// POUs/System/SystemInfo
{attribute 'no_check'}
//Provides all information of PlcAppSystemInfo plus addtional infos like time stamps from various source and in different formats
//
//PlcAppSystemInfo -> https://infosys.beckhoff.com/english.php?content=../content/1033/globaldatatypes/9007199969559691.html&id=7934476013631172214
//TwimCAT time sources -> https://infosys.beckhoff.com/english.php?content=../content/1033/ethercatsystem/2469114379.html&id=
//
FUNCTION_BLOCK SystemInfo
VAR_OUTPUT CONSTANT
{attribute 'displaymode':='binary'}
	OPTION_US_DATE_FORMAT									:	BYTE := 2#0000_0001; //Enable US date format in time stamp - mm/dd/yy
{attribute 'displaymode':='binary'}
	OPTION_US_TIME_FORMAT									:	BYTE := 2#0000_0010; //Enable time in US format - AM/PM vs 24h
{attribute 'displaymode':='binary'} 
	OPTION_TIME_STR_ADD_MS									:	BYTE := 2#0000_0100; //Add ms to time string 
{attribute 'displaymode':='binary'} 
	OPTION_DISABLE_DEV_IDENT								:	BYTE := 2#0000_1000; //Disable to read device identification during boot up (Call FB_GetDeviceIdentificationEx)
END_VAR                     								
VAR_INPUT                   						
	Enable													:	BOOL := TRUE; //Enable function block
	ResetTrig												:	BOOL := FALSE; //Reset Old boot data fault signal
	RtcSyncCylce											:	DWORD := 60; //in seconds - see documentation for "FB_LocalSystemTime"
	KeepOutputsOnBP 										: 	BOOL := FALSE; //The flag can be set to avoid that the outputs are zero-filled if a breakpoint is reached. The task keeps running. Only the execution of PLC code is interrupted.
{attribute 'displaymode':='binary'}
	Options													:	BYTE := 2#0000_0000; //option constants are alreay predefined, so they can accordingly be passed symbolically to the block 
	DateStrSeperator										:	STRING(1) := '/';
END_VAR
VAR_OUTPUT
//PlcAppSystemInfo and cycle time inforamtion from caller task 
	ObjId													: 	OTCID; //Object ID of the PLC project instance
	AdsPort 												: 	UINT; //ADS port of PLC application 
	TComSrvPtr 												: 	ITComObjectServer; // Pointer to TcCOM Object Server 
	AppName													: 	STRING(63); //TwinCAT generated name containing the port number. 
	ProjectName 											: 	STRING(63); //The name of the PLC project. 
	AppTimestampDT											:	DT; //Date and time of application start 
	AppTimestamp											:	STRING(25);	//Date and time of application start in string format
	TaskIndex												:	INT ; //Task index of SysInfo caller
	TaskCnt													: 	UDINT; //The number of tasks in the actual runtime system
	
	Flags 													: 	DWORD; //Boot flags
	LicensesPending 										: 	BOOL;
	BSODOccured 											: 	BOOL;										
	BootDataLoaded											: 	BOOL;//PERSISTENT variables: LOADED (without error)
	OldBootData												: 	BOOL; //PERSISTENT variables: INVALID (the back-up copy was loaded, since no valid data was present)
	NoBootDataLoaded										:	BOOL; //Error no boot data loaded
//	PersistentStatus 										: 	EPlcPersistentStatus;

	LoggedIn												:	BOOL;
	ShutdownInProgress 										: 	BOOL;	
	OnlineChangeCount										: 	UDINT; //The number of online changes made since the last complete download.
	OnlineChange											:	BOOL; //Online change count changed since last plc cycle

{attribute 'displaymode':='hex'}
	CpuCounter												:	ULINT;
	CycleTime         										: 	UDINT;//Cylce time read from PlcAppSystemInfo in multiples of 100 ns.
	CycleTimeNS         									: 	UDINT;//Cylce time in nanoseconds
	CycleTimeT       										: 	TIME; //Cycle time in time format
	CycleTimeLT       										: 	LTIME; //Cycle time in ltime format
	CycleTimeFloat											:	LREAL;//Cycle time in float format <s.ms>

	DevIdentValid											:	BOOL;
	pDevIdent												:	POINTER TO ST_DeviceIdentificationEx := ADR(InstGetDevIdent.stDevIdent);
	
//General	
	TimezoneId												: 	E_TimeZoneID;
	TimeZoneInfo											:	ST_TimeZoneInformation; //Provides actual time zone and bias from local time to UTC e.g. UTC=MEC-01:00 (-60min from lcoal MEZ in Standard time to UTC)
	MonthDays												:	WORD;
	LeapYear												:	BOOL;
	DayOfYear												:	WORD;
	WeekOfYear												:	WORD;
	UtcTimeFT												:	Tc2_Utilities.T_FILETIME; //Current UTC System/TwinCAT time T_FILETIME format, structure representing a 64-bit value with the a number of 100-nanosecond intervals since January 1, 1601 (UTC) (dwLowDateTime : DWORD / dwHighDateTime : DWORD)
//	UtcTimeFT												:	Tc2_Utilities.T_FILETIME64; //Current UTC System/TwinCAT time T_FILETIME format, structure representing a 64-bit value with the a number of 100-nanosecond intervals since January 1, 1601 (UTC) (dwLowDateTime : DWORD / dwHighDateTime : DWORD)
	UtcTimeSTRUCT											:	Tc2_Utilities.TIMESTRUCT; //Current UTC System/TwinCAT time in TIMESTRUCT format
	UtcTimezoneBias											:	DINT;   //Bias from UTC to local time in minutes e.g. MEZ=UTC+01:00 (60min)  
	TimeDT													:	DATE_AND_TIME;	//Current time in DATE_AND_TIME format: DT#1970-01-01-00:00 -> DT#2106-02-06-06:28:15
//	TimeLDT													:	LDATE_AND_TIME;	//Current time in 64bit LDATE_AND_TIME format: DT#1970-01-01-00:00 -> DT#2262-4-10-23:59:59.99999999
	TimeTOD													:	TOD; //Current time in TOD format, range from TOD#00:00 -> TOD#1193:02:47.295
	TimeFT													:	Tc2_Utilities.T_FILETIME; //Current time in T_FILETIME format, structur representing a 64-bit value with the a number of 100-nanosecond intervals since January 1, 1601 (UTC) (dwLowDateTime : DWORD / dwHighDateTime : DWORD)
//	TimeFT													:	Tc2_Utilities.T_FILETIME64; //Current time in T_FILETIME format, structur representing a 64-bit value with the a number of 100-nanosecond intervals since January 1, 1601 (UTC) (dwLowDateTime : DWORD / dwHighDateTime : DWORD)
	TimeSTRUCT												:	Tc2_Utilities.TIMESTRUCT; //Current time in TIMESTRUCT format
	Datestamp												:	DATE; //D#1970-01-01 -> D#2106-02-06
	DateStr													:	STRING(15);	(* dd.mm.jj or mm.dd.jj *)	
	TimeStr													:	STRING(15);	(* hh:mm:ss.xxx or hh:mm:ss.xxxPM/AM *)
	TimeStamp												:	STRING(25); (* DateStr + TimeStr *)	
	TimeStamp2												:	STRING(25); (* YYYY-MM-DDTHHMMSS for example YYYY-MM-DD_HHMMSS_Name.txt *)
	TimeStamp3												:	STRING(25); (* YYYY-MM-DD-hh:mm:ss.xxx *)
	DateStrISO												:	STRING(15);	(* jjjj-mm-dd *)
	TimeStrISO												:	STRING(15);	(* hh:mm:ss *)
	TimeStrISO2												:	STRING(15);	(* hh:mm:ss.xxx *)	
	TimeStampIso											:	STRING(30);	(* jjjj-mm-dd'T'hh:mm:ss.xxx local time*)	
//	TimeStampIsoZulu										:	STRING(30);	(* jjjj-mm-dd'T'hh:mm:ss.xmsZ - Iso timestamp in UTC (ZULU)*)	
//	TimeStampIsoUtc											:	STRING(30);	(* jjjj-mm-dd'T'hh:mm:ss.xms+mm:ss - Iso timestamp with UTC offset *)	

	TimeStampStartup										:	DATE_AND_TIME; //Timestamp of startup
	DCTime													:	Tc2_EtherCAT.T_DCTIME64; //Current TwinCAT distributed clock time in 64-bit T_DCTIME64 format. The smallest unit is a nanosecond.
	DCTimeSTRUCT											:	Tc2_Utilities.TIMESTRUCT;//Current TwinCAT distributed clock time in TIMESTRUCT format
//	SysTimeFT												:	Tc2_Utilities.T_FILETIME64; //Current UTC System/TwinCAT time T_FILETIME format, structure representing a 64-bit value with the a number of 100-nanosecond intervals since January 1, 1601 (UTC) (dwLowDateTime : DWORD / dwHighDateTime : DWORD)
	SysTimeFT												:	Tc2_Utilities.T_FILETIME; //Current UTC System/TwinCAT time T_FILETIME format, structure representing a 32-bit value since January 1, 1601 (UTC) (dwLowDateTime : DWORD / dwHighDateTime : DWORD)
	SysTimeSTRUCT											:	Tc2_Utilities.TIMESTRUCT; //Current UTC System/TwinCAT time in TIMESTRUCT format
	
END_VAR
VAR
	(* Inst. Get Taskindex *)
	InstGETCURTASKINDEX										: 	GETCURTASKINDEX;
	InstLocalSystemTime										:	FB_LocalSystemTime;
	InstNtSetLocalTime										:	NT_SetLocalTime := (NETID := '', TMOUT := DEFAULT_ADS_TIMEOUT);
	InstTimeZoneInfo										:	FB_GetTimeZoneInformation;
	InstCpuCouter											:	GETCPUCOUNTER;
	InstSystemTime											:	GetSystemTime;
	
	
	InstGetDevIdent											:	FB_GetDeviceIdentificationEx;
	_OnlineChangeCount										: 	UDINT; 
	_sec													:	WORD;
	_hour													:	WORD;
	_day													:	WORD;
	_Init													:	BOOL;
END_VAR

	(* Evaluate the PlcAppSystemInfo and and get sytstem timestamp					*)
	(********************************************************************************)
	
(* Get Current Task Index ************************************************************************)
	IF InstGETCURTASKINDEX.index = 0 then InstGETCURTASKINDEX(index => TaskIndex); END_IF

(* Read System Info Current Task *****************************************************************)	
	(* Get static information and boot error messages *)
	IF TwinCAT_SystemInfoVarList._TaskInfo[InstGETCURTASKINDEX.Index].FirstCycle 
	THEN
		AppTimestampDT										:= TwinCAT_SystemInfoVarList._AppInfo.AppTimestamp;
		AppTimestamp										:= DT_TO_STRING(AppTimestampDT);
		AppTimestamp										:= DELETE(AppTimestamp,3,1);
			
		TaskIndex											:= InstGETCURTASKINDEX.Index;
		TaskCnt 											:= TwinCAT_SystemInfoVarList._AppInfo.TaskCnt;
		
		ObjId												:= TwinCAT_SystemInfoVarList._AppInfo.ObjId;
		AppName												:= TwinCAT_SystemInfoVarList._AppInfo.AppName;	
		ProjectName											:= TwinCAT_SystemInfoVarList._AppInfo.ProjectName;	
		AdsPort												:= TwinCAT_SystemInfoVarList._AppInfo.AdsPort;	
			
		Flags												:= TwinCAT_SystemInfoVarList._AppInfo.Flags;
//		PersistentStatus									:= TwinCAT_SystemInfoVarList._AppInfo.PersistentStatus;
		
		BootDataLoaded										:= TwinCAT_SystemInfoVarList._AppInfo.BootDataLoaded;
		OldBootData											:= TwinCAT_SystemInfoVarList._AppInfo.OldBootData;
		NoBootDataLoaded									:= NOT BootDataLoaded AND NOT OldBootData;
		BSODOccured 										:= TwinCAT_SystemInfoVarList._AppInfo.BSODOccured;
		
		CycleTime         									:= TwinCAT_SystemInfoVarList._TaskInfo[TaskIndex].CycleTime;
		CycleTimeNS         								:= TwinCAT_SystemInfoVarList._TaskInfo[TaskIndex].CycleTime * 100;
		CycleTimeT											:= LREAL_TO_TIME(UDINT_TO_LREAL(CycleTime) * 0.0001 );
		CycleTimeLT											:= TO_LTIME(CycleTimeNS);	
		CycleTimeFloat										:= (UDINT_TO_LREAL(CycleTime) * 0.0001 / 1000.0);	
		
	ELSIF ResetTrig
	THEN
		resetBootInfo();
	ELSIF NOT Enable
	THEN
		RETURN;
	END_IF
	
	OnlineChangeCount										:= TwinCAT_SystemInfoVarList._AppInfo.OnlineChangeCnt;
	OnlineChange											:= _OnlineChangeCount <> OnlineChangeCount;
	_OnlineChangeCount										:= OnlineChangeCount;
	LoggedIn 												:= TwinCAT_SystemInfoVarList._AppInfo.LoggedIn;
	ShutdownInProgress 										:= TwinCAT_SystemInfoVarList._AppInfo.ShutdownInProgress;
	LicensesPending 										:= TwinCAT_SystemInfoVarList._AppInfo.LicensesPending;
	TComSrvPtr												:= TwinCAT_SystemInfoVarList._AppInfo.TComSrvPtr;
	TwinCAT_SystemInfoVarList._AppInfo.KeepOutputsOnBP		:= KeepOutputsOnBP;		

(* CPU System counter ****************************************************************************)
	InstCpuCouter(cpuCntLoDW => CpuCounter);	
	MEMCPY(ADR(CpuCounter) + SIZEOF(InstCpuCouter.cpuCntHiDW),ADR(InstCpuCouter.cpuCntHiDW),SIZEOF(InstCpuCouter.cpuCntHiDW));
	
(* Get device identification structure ***********************************************************)
	InstGetDevIdent(
		bExecute	:= NOT Options.3, 
		tTimeout	:= , 
		sNetId		:= , 
		bBusy		=> , 
		bError		=> , 
		nErrorID	=> , 
		stDevIdent	=> );	
	pDevIdent												:= ADR(InstGetDevIdent.stDevIdent);
	IF NOT InstGetDevIdent.bBusy
	THEN
		DevIdentValid										:= NOT InstGetDevIdent.bError;
		
		IF InstGetDevIdent.bError AND ResetTrig
		THEN
			InstGetDevIdent(bExecute := FALSE);			
		END_IF
	ELSE	
		DevIdentValid										:= FALSE;
	END_IF
	
(* Read timezone information every day time ******************************************************)
	IF Enable AND NOT InstTimeZoneInfo.bExecute
		OR InstTimeZoneInfo.bBusy
	THEN
		InstTimeZoneInfo(
			sNetID	:= , 
			bExecute:= TRUE, 
			tTimeout:= , 
			bBusy	=> , 
			bError	=> , 
			nErrID	=> , 
			tzID	=> TimeZoneId, 
			tzInfo	=> TimeZoneInfo);
		IF NOT InstTimeZoneInfo.bBusy 
		THEN
			CASE TimeZoneId OF 
			eTimeZoneID_Invalid:	UtcTimezoneBias			:= 0;				
			eTimeZoneID_Standard:	UtcTimezoneBias			:= -1 * (TimeZoneInfo.bias + TimeZoneInfo.standardBias);
			eTimeZoneID_Daylight:	UtcTimezoneBias			:= -1 * (TimeZoneInfo.bias + TimeZoneInfo.daylightBias);
			ELSE //eTimeZoneID_Unknown:		
				UtcTimezoneBias								:= 0;	
			END_CASE
		END_IF
	ELSIF NOT Enable AND InstTimeZoneInfo.bExecute 
		OR InstTimeZoneInfo.bError AND ResetTrig
	THEN
		InstTimeZoneInfo(bExecute:= FALSE);
	END_IF
		
(* Actual EtherCAT DC time in DCTIME64 format ****************************************************************)
	DCTime													:= F_GetActualDcTime64();
	DCTimeSTRUCT											:= DCTIME64_TO_SYSTEMTIME(DCTime);

(* Get TwinCAT/system time according to system time zone initialized during TC start ******************************************************)
	InstSystemTime(timeHiDW => UtcTimeFT.dwHighDateTime,timeLoDW => UtcTimeFT.dwLowDateTime );
	SysTimeSTRUCT											:= FILETIME_TO_SYSTEMTIME(UTCTimeFT);	
	
//	SysTimeFT												:= F_GetSystemTime();	 
//	SysTimeSTRUCT											:= FILETIME64_TO_SYSTEMTIME(UTCTimeFT);	 
	
(* evalutate systemtime ************************************************************************)
	InstLocalSystemTime(
		sNetID		:= '',
		bEnable		:= Enable,
		dwCycle		:= SEL(InstNtSetLocalTime.START, RtcSyncCylce, 1), //Short update cylce to read windows time after it was set
		dwopt		:= (* Default *),
		tTimeout	:= (* Default *),
		bValid		=> ,
		systemTime	=> TimeSTRUCT,
		tzID		=> );

(* Get TwinCAT/system time in UTC Filetime format ******************************************************)
	IF InstLocalSystemTime.bValid 
	THEN				
		//Update cyclic
//		TimeFT												:= SYSTEMTIME_TO_FILETIME64(TimeSTRUCT);
		TimeFT												:= SYSTEMTIME_TO_FILETIME(TimeSTRUCT);
		TimeDT 												:= SYSTEMTIME_TO_DT(TimeSTRUCT);
//		TimeLDT												:= SYSTEMTIME_TO_LDT(TimeSTRUCT);	
		TimeStamp3											:= SYSTEMTIME_TO_STRING(TimeSTRUCT);
		TimeTOD												:= SEL(Options.2 ,TO_TOD(TimeDT)  , DWORD_TO_TOD(TO_DWORD(TO_TOD(TimeDT)) + TimeSTRUCT.wMilliseconds));  
		TimeStrISO											:= DELETE(TO_STRING(TimeTOD),4,1);

		IF TimeSTRUCT.wMilliseconds < 10 
		THEN
			TimeStrISO2 									:= CONCAT(TimeStrISO,CONCAT('.00',WORD_TO_STRING(TimeSTRUCT.wMilliseconds)));
		ELSIF TimeSTRUCT.wMilliseconds < 100
		THEN
			TimeStrISO2 									:= CONCAT(TimeStrISO,CONCAT('.0',WORD_TO_STRING(TimeSTRUCT.wMilliseconds)));			
		ELSE        										
			TimeStrISO2 									:= CONCAT(TimeStrISO,CONCAT('.',WORD_TO_STRING(TimeSTRUCT.wMilliseconds)));	
		END_IF 	
		
		TimeStampISO										:= CONCAT(DateStrISO , CONCAT('T',TimeStrISO2));
				
		UtcTimeFT											:= F_TranslateFileTimeBias(TimeFT,UtcTimezoneBias,TRUE);
		UtcTimeSTRUCT										:= FILETIME_TO_SYSTEMTIME(UTCTimeFT);	
//		UtcTimeFT											:= F_TranslateFileTime64Bias(TimeFT,UtcTimezoneBias,TRUE);
//		UtcTimeSTRUCT										:= FILETIME64_TO_SYSTEMTIME(UTCTimeFT);	

//		TimeStampIsoZulu									:= SYSTEMTIME_TO_ISO8601(UtcTimeSTRUCT,0,FALSE,3);
//		TimeStampIsoZulu									:= CONCAT(DELETE(TimeStampIsoZulu,6,24),'Z');
//		TimeStampIsoUtc										:= SYSTEMTIME_TO_ISO8601(UtcTimeSTRUCT,TO_INT(UtcTimezoneBias),TRUE,3);
	
		//Create time format
		IF Options.1
		THEN (* US time format hh.mm.ss AM/PM ***************)
			IF TimeSTRUCT.wHour < 10 
			THEN
				TimeStr 									:= CONCAT('0',WORD_TO_STRING(TimeSTRUCT.wHour));
			ELSIF TimeSTRUCT.wHour > 12 
			THEN
				TimeStr 									:= WORD_TO_STRING(TimeSTRUCT.wHour - 12);
				IF TimeSTRUCT.wHour - 12 < 10
				THEN
					TimeStr									:= CONCAT('0',TimeStr);
				END_IF
			ELSE         									
				TimeStr 									:= WORD_TO_STRING(TimeSTRUCT.wHour);
			END_IF		                                    
		ELSE  (* Time hh.mm.ss.xxms ***************)          
			IF TimeSTRUCT.wHour < 10                        
			THEN                                            
				TimeStr 									:= CONCAT('0',WORD_TO_STRING(TimeSTRUCT.wHour));
			ELSE        									
				TimeStr 									:= WORD_TO_STRING(TimeSTRUCT.wHour);
			END_IF			
		END_IF
		
		TimeStr 											:= CONCAT(TimeStr,':');
		
		IF TimeSTRUCT.wMinute < 10 
		THEN
			TimeStr 										:= CONCAT(TimeStr,CONCAT('0',WORD_TO_STRING(TimeSTRUCT.wMinute)));
		ELSE
			TimeStr 										:= CONCAT(TimeStr,WORD_TO_STRING(TimeSTRUCT.wMinute));
		END_IF
		
		TimeStr 											:= CONCAT(TimeStr,':');
		
		IF TimeSTRUCT.wSecond < 10 
		THEN
			TimeStr 										:= CONCAT(TimeStr,CONCAT('0',WORD_TO_STRING(TimeSTRUCT.wSecond)));
		ELSE        										
			TimeStr 										:= CONCAT(TimeStr,WORD_TO_STRING(TimeSTRUCT.wSecond));
		END_IF  
												
		IF Options.2
		THEN //add ms to timestamp
			TimeStr 										:= CONCAT(TimeStr,'.');
			TimeStr 										:= CONCAT(TimeStr,WORD_TO_STRING(TimeSTRUCT.wMilliseconds));
		END_IF
		
		IF Options.1
		THEN //US time format
			TimeStr 										:= CONCAT(TimeStr,SEL(TimeSTRUCT.wHour > 12,' AM', ' PM'));
		END_IF
		
		(* TimeStamp Format DE: DD.MM.YY-Stunde:Minute:Sekunde.xxx,*)
		TimeStamp 											:= CONCAT(DateStr,'-');
		TimeStamp 											:= CONCAT(TimeStamp,TimeStr);
		
		IF _hour <> TimeSTRUCT.wHour OR NOT _Init
		THEN
			_Hour											:= TimeSTRUCT.wHour;		
			//Create date in US fromat with seperator / ************************************************
			IF Options.0
			THEN (* Date mm/dd/jj ********************)
				IF TimeSTRUCT.wMonth < 10 
				THEN
					DateStr 								:= CONCAT('0',WORD_TO_STRING(TimeSTRUCT.wMonth));
				ELSE        								
					DateStr 								:= WORD_TO_STRING(TimeSTRUCT.wMonth);
				END_IF		                                
				DateStr 									:= CONCAT(DateStr,DateStrSeperator);
				IF TimeSTRUCT.wDay < 10                     
				THEN                                        
					DateStr 								:= CONCAT(DateStr,CONCAT('0',WORD_TO_STRING(TimeSTRUCT.wDay)));
				ELSE        								
					DateStr 								:= CONCAT(DateStr,WORD_TO_STRING(TimeSTRUCT.wDay));
				END_IF                                      
															
				DateStr 									:= CONCAT(DateStr,DateStrSeperator);
				DateStr 									:= CONCAT(DateStr,RIGHT(WORD_TO_STRING(TimeSTRUCT.wYear),2));		
		                                                    
			ELSE (* Date dd.mm.jj ********************)	    
				IF TimeSTRUCT.wDay < 10                     
				THEN                                        
					DateStr 								:= CONCAT('0',WORD_TO_STRING(TimeSTRUCT.wDay));
				ELSE        								
					DateStr 								:= WORD_TO_STRING(TimeSTRUCT.wDay);
				END_IF                                      
				DateStr 									:= CONCAT(DateStr,DateStrSeperator);
				IF TimeSTRUCT.wMonth < 10                   
				THEN                                        
					DateStr 								:= CONCAT(DateStr,CONCAT('0',WORD_TO_STRING(TimeSTRUCT.wMonth)));
				ELSE        								
					DateStr 								:= CONCAT(DateStr,WORD_TO_STRING(TimeSTRUCT.wMonth));
				END_IF                                      
															
				DateStr 									:= CONCAT(DateStr,DateStrSeperator);
				DateStr 									:= CONCAT(DateStr,RIGHT(WORD_TO_STRING(TimeSTRUCT.wYear),2));	
			END_IF      

			DateStrISO										:= DELETE(TO_STRING(TO_DATE(TimeDT)),2,1);
			
			(* information of year *)                       
			MonthDays										:= F_GetMaxMonthDays(TimeSTRUCT.wYear,TimeSTRUCT.wMonth);
			LeapYear										:= F_YearIsLeapYear(TimeSTRUCT.wYear) ;
			WeekOfYear										:= F_GetWeekOfTheYear(TimeDT);
			DayOfYear										:= F_GetDOYOfYearMonthDay(TimeSTRUCT.wYear,TimeSTRUCT.wMonth,TimeSTRUCT.wDay);
			DateStamp										:= TO_DATE(TimeDT);		
			
			IF NOT _INIT AND_THEN TO_DINT(TimeStampStartup) = 0  
			THEN					
				TimeStampStartup							:= SYSTEMTIME_TO_DT(TimeSTRUCT);
			END_IF
			
			IF NOT InstTimeZoneInfo.bBusy THEN InstTimeZoneInfo(bExecute:= FALSE); END_IF

            _INIT											:= TRUE;            
		END_IF //hour
		
		IF _sec <> TimeSTRUCT.wSecond 
		THEN	
			_sec 											:= TimeSTRUCT.wSecond;
														
			(* TimeStamp2 FileName YYYY-MM-DD_HHMMSS *)
			TimeStamp2										:= CONCAT(DateStrISO , '_');
			IF TimeSTRUCT.wHour < 10                    	
			THEN                                        	
				TimeStamp2 									:= CONCAT(TimeStamp2,CONCAT('0',WORD_TO_STRING(TimeSTRUCT.wHour)));
			ELSE           									
				TimeStamp2 									:= CONCAT(TimeStamp2,WORD_TO_STRING(TimeSTRUCT.wHour));
			END_IF                                      	
			IF TimeSTRUCT.wMinute < 10                  	
			THEN                                        	
				TimeStamp2 									:= CONCAT(TimeStamp2,CONCAT('0',WORD_TO_STRING(TimeSTRUCT.wMinute)));
			ELSE           									
				TimeStamp2 									:= CONCAT(TimeStamp2,WORD_TO_STRING(TimeSTRUCT.wMinute));
			END_IF                                      	
			IF TimeSTRUCT.wSecond < 10                  	
			THEN                                        	
				TimeStamp2 									:= CONCAT(TimeStamp2,CONCAT('0',WORD_TO_STRING(TimeSTRUCT.wSecond)));
			ELSE           									
				TimeStamp2 									:= CONCAT(TimeStamp2,WORD_TO_STRING(TimeSTRUCT.wSecond));
			END_IF
		END_IF //second update
													
	END_IF

(* set system time *****************************************************************************)
	InstNtSetLocalTime(
		NETID		:= , 
		TIMESTR		:= , 
		START		:= , // Start by Methode "SetSysTime" 
		TMOUT		:= , 
		BUSY		=> , 
		ERR			=> ); 
	
	IF InstNtSetLocalTime.START AND NOT InstNtSetLocalTime.BUSY
	THEN //Take care that all timestamp get updated after set a new time
		InstNtSetLocalTime.START							:= FALSE;	
		_Init												:= FALSE;								
	END_IF
	
(**************************************************************************************************)

PROPERTY PUBLIC actDCTimeWithTimezoneBias : T_DCTIME64
GET
actDCTimeWithTimezoneBias							:= F_GetActualDcTime64() + (TO_ULINT(UtcTimezoneBias) * 60 * EC_DCTIME_TICKSPERSEC64);
END_GET
END_PROPERTY

PROPERTY PUBLIC optAddmsToTimeString : BOOL
GET
optAddmsToTimeString := Options.2;
END_GET
SET
Options.2 := optAddmsToTimeString;
END_SET
END_PROPERTY

PROPERTY PUBLIC  optDisableReadDeviceIdentification : BOOL
GET
optDisableReadDeviceIdentification := Options.3;
END_GET
SET
Options.3 := optDisableReadDeviceIdentification;
END_SET
END_PROPERTY

PROPERTY PUBLIC optEnableUSDateFormat : BOOL
GET
optEnableUSDateFormat := Options.0;
END_GET
SET
Options.0 := optEnableUSDateFormat;
END_SET
END_PROPERTY

PROPERTY PUBLIC optEnableUSTimeFormat : BOOL
GET
optEnableUSTimeFormat := Options.1;
END_GET
SET
Options.1 := optEnableUSTimeFormat;
END_SET
END_PROPERTY

METHOD PUBLIC resetBootInfo : BOOL  //Return value = TRUE if execution finished
VAR_INPUT
END_VAR
OldBootData 												:= FALSE;
BSODOccured													:= FALSE;
NoBootDataLoaded											:= FALSE;
resetBootInfo												:= TRUE;
END_METHOD

METHOD PUBLIC setSysTime  : BOOL //Return value = TRUE if execution finished
VAR_INPUT
	TimeStruct		: TIMESTRUCT;
END_VAR
InstNtSetLocalTime(
		NETID		:= '', 
		TIMESTR		:= TimeStruct, 
		START		:= NOT InstNtSetLocalTime.START AND TimeStruct.wYear > 2000 
						AND TimeStruct.wDay > 0 AND TimeStruct.wMonth	< 32	
						AND TimeStruct.wMonth > 0 AND TimeStruct.wMonth	< 13	
						AND TimeStruct.wHour >= 0 AND TimeStruct.wHour	< 24	
						AND TimeStruct.wMinute >= 0 AND TimeStruct.wMinute < 60
						AND TimeStruct.wSecond >= 0 AND TimeStruct.wSecond < 60				
						OR InstNtSetLocalTime.BUSY, 
		TMOUT		:= , 
		BUSY		=> , 
		ERR			=> , 
		ERRID		=> );
		
setSysTime													:= InstNtSetLocalTime.BUSY;
END_METHOD

END_FUNCTION_BLOCK

// POUs/Fieldbus/EtherCAT/EcDiagBase
{attribute 'no_check'}
FUNCTION_BLOCK EcDiagBase
VAR_OUTPUT CONSTANT         								
	MIN_SLAVES												: 	UINT := 1;
	MAX_SLAVES												: 	UINT := PARAM.ETHERCAT_DIAG_MAX_SLAVES;	//EC_MAX_SLAVES = 65535 Slaves;
END_VAR
VAR_INPUT
	Enable													:	BOOL := TRUE;//FB will be processed as long as enable is TRUE 
	
	DelReadSlavesDiag										:	TIME := T#2S; //Damping time to read diagnostic if error is detected 
(* Components *)            								
	IO														:	EcMasterIO;
END_VAR                     								
VAR_OUTPUT                  								
	MasterOK												:	BOOL; 	//TRUE when Master/EtherCAT is OK
	SlavesOK												:	BOOL;	//TRUE if no slave is in error state
	NoOfSlavesNOK											:	UINT;
	NoOfMissedSlaves										:	INT; //No of slaves missed incl. hot connect slaves 
	NoOfHotConnectGroups									:	UINT;
	NoOfHotConnectSlaves									:	UINT;
	
	pSlaveInfoData											:	POINTER TO ARRAY [MIN_SLAVES..MAX_SLAVES] OF EC_SLAVE_DIAG_INFO_DATA := ADR(SlavesDiag.InfoData); //configured slaves			
	DiagBusy												:	BOOL;
	ErrorReadDiag											:	BOOL;
END_VAR
VAR
(* Local  ***********************************************************)
	MemSlaveCount											:	UINT;
	MemDevState												:	UINT;
	InitDone												:	BOOL;
	
(* trigger ********************************************************)
	rtReadDiag												: r_Trig;

(* Timer **********************************************************)
	tonDelTrigDiag											:	ton;

(* events *********************************************************)

(* function-block *************************************************)
	SlavesDiag												:	EcSlavesDiag;
	
(* dummy **********************************************************)
	idx,i													:	INT;											
END_VAR

(* Base diagnostic of EtherCAT 					*)
(************************************************)

(* Work IO *************************************************)
	IO();

(* trigger slaves diag *************************************************************)
	IF NOT tonDelTrigDiag.IN AND NOT SlavesDiag.Busy
		AND( 
		IO.FramesWcStateChanged
		OR MemDevState <> IO.DevState
		OR MemSlaveCount <> IO.SlaveCountTotal
		OR NoOfSlavesNOK > 0 
		OR NOT InitDone)
	THEN
		tonDelTrigDiag(IN := TRUE , PT := DelReadSlavesDiag);
	END_IF
	//Run delay	
	tonDelTrigDiag();
	
	rtReadDiag(CLK := Enable AND tonDelTrigDiag.Q);
	IF SlavesDiag.Error
	THEN
		adsLogError('Error in FB EcSlavesDiag: %s',  SlavesDiag.ErrorText);
	ELSIF rtReadDiag.Q 
	THEN 	
		tonDelTrigDiag(IN := FALSE); //Restart timer
		SlavesDiag.optReadScannedSlaves						:= MemSlaveCount <> IO.SlaveCountTotal OR NoOfMissedSlaves > 0 OR NoOfSlavesNOK > 0 OR SlavesDiag.InvalidVPRS; //Scan slaves if invalid VPRS or HC groups are configured
	//	SlavesDiag.optSortInfoData 							:= ;
	//	SlavesDiag.optUpdateTopoData						:= ;
	//	SlavesDiag.optUpdateConfigData 						:= ;
		
	 	MemSlaveCount 										:= IO.SlaveCountTotal;
		MemDevState 										:= IO.DevState;
		InitDone											:= TRUE;
	END_IF
	SlavesDiag(Execute := rtReadDiag.Q ,MasterAmsNetId := IO.AmsNetIdStr, NoOfSlavesNOK => NoOfSlavesNOK, NoOfHCGroups => NoOfHotConnectGroups, NoOfHCSlaves => NoOfHotConnectSlaves, Busy => DiagBusy , Error => ErrorReadDiag);		
	pSlaveInfoData											:= ADR(SlavesDiag.InfoData);
		
(***********************************************************************************)
	MasterOK 												:= IO.DevStateBits.NoError;
	SlavesOK												:= MasterOK AND SlavesDiag.NoOfSlavesNOK = 0;
	NoOfMissedSlaves										:= TO_INT(IO.CfgSlaveCount) - TO_INT(IO.SlaveCountTotal);
	
(*********************************************************************************)

END_FUNCTION_BLOCK

// POUs/Logging/adsLogError
{attribute 'no_check' := ''}
//Writes a string as a error message into the TwinCAT AMS Logger and Windows Event Log with an possible argument
//Please see Beckhoff information system "ADSLOGxxxx" for detailed information.
//Intention of this function is to use the handy ADSLOGxxxx with a predefined msgCtrlMask of "ADSLOG_MSGTYPE_STRING OR ADSLOG_MSGTYPE_HINT OR ADSLOG_MSGTYPE_LOG"
FUNCTION adsLogError : DINT //Write error message into ADS log windows - Return value will be error code or 0 if OK
VAR_INPUT               											
	MsgFmtStr												:	T_MaxString; //Message text with %s as placeholder for StrArg
(*	dintArg													:	DINT; //DINT argument for message - to be replaced by %d *) 
	StrArg													:	T_MaxString; //String argument for message - to be replaced by %s
(*	realArg													:	LREAL; //LREAL argument for message - to be replaced by %f *) 
END_VAR
VAR
	msgCtrlMask												:	DWORD; (* 	ADSLOG_MSGTYPE_HINT Meldungstyp ist Hinweis.
																				ADSLOG_MSGTYPE_WARN Meldungstyp ist Warnung.  
																				ADSLOG_MSGTYPE_ERROR Meldungstyp ist Fehler.  
																				ADSLOG_MSGTYPE_LOG Meldung wird in das Logbuch geschrieben.  
																				ADSLOG_MSGTYPE_MSGBOX Meldung wird in einer Messagebox ausgegeben.  
																				ADSLOG_MSGTYPE_RESOURCE Meldung wird aus einer Ressource-Datei geholt. (wird momentan nicht  unterstützt)  
																				ADSLOG_MSGTYPE_STRING 	Meldung ist direkt angegebener String (default).  *)	
END_VAR

(* create fixed message ctrl mask **********************************)
	msgCtrlMask												:= ADSLOG_MSGTYPE_STRING OR ADSLOG_MSGTYPE_ERROR OR ADSLOG_MSGTYPE_LOG;

(* write string which includes a floating-number ******************)
(*	AdsLogError 											:= ADSLOGLREAL(msgCtrlMask, msgFmtStr, realArg); *)
	
(* write string which includes a DINT-number *******************)
(*	AdsLogError 											:= ADSLOGDINT(msgCtrlMask, msgFmtStr, dintArg); *)

(* write string which includes an other string e.g. 'hallo: %s what's up' ***************)
	adsLogError 											:= ADSLOGSTR(msgCtrlMask, msgFmtStr,strArg); 

(*****************************************************)

END_FUNCTION

// POUs/Fieldbus/EtherCAT/EcDiagBase_wEvents
{attribute 'no_check'}
FUNCTION_BLOCK EcDiagBase_wEvents EXTENDS EcDiagBase
VAR_OUTPUT CONSTANT         								
END_VAR
VAR_INPUT
	ConfirmTrig												:	BOOL;
	SourceId												: 	UDINT := 103000; //Multisource id 
END_VAR                     								
VAR_OUTPUT                  								
	{attribute 'displaymode':='binary'}
	EventStatus												:	DWORD;
END_VAR
VAR
(* Local  ***********************************************************)

	
(* trigger ********************************************************)


(* Timer **********************************************************)


(* events *********************************************************)
	Event													:	EventHandlingGrp10;
	
(* function-block *************************************************)

	
(* dummy **********************************************************)
										
END_VAR

(* Base diagnostic of EtherCAT with events		*)
(************************************************)

(* Call super  *************************************************)
	SUPER^();
	
(* Fire events **********************************************************************)
	_callEvents();
	
(**************************************************************************************)

METHOD PRIVATE _callEvents : BOOL
VAR_INPUT
END_VAR
(* Events anzeigen ***************************************************)
	(* Init events *)
	IF Event.no[1].Text1 <> IO.Name
	THEN
		FOR i := Event.MIN_EVENT TO Event.MAX_EVENT 
		DO
			Event.no[i].Text1								:= IO.Name;
		END_FOR
	END_IF 

	(* Master Error Event *)
	
	Event.no[1].Flag										:= NOT IO.DevStateBits.NoError AND NOT IO.DevStateChanged AND NOT ConfirmTrig;
	Event.no[1].pText3										:= ADR(IO.DevStateText);

	(* Error Port Link *)
	Event.no[2].Flag										:=(NOT IO.LinkOK_PortA OR NOT IO.LinkOK_PortB) AND NOT SlavesDiag.Busy AND NOT tonDelTrigDiag.IN;
	IF Event.no[2].Flag
	THEN
		Event.no[2].Text2									:= TO_STRING(NoOfMissedSlaves);
		Event.no[2].pText3									:= ADR(SlavesDiag.FirstErrorSlave.ConfigName);	
	END_IF

	(* No Slave Com *)
	Event.no[3].Flag										:= IO.AllFramesMissing AND NoOfMissedSlaves = 0 AND NOT IO.DevStateChanged AND NOT SlavesDiag.Busy AND NOT tonDelTrigDiag.IN;
	IF Event.no[3].Flag
	THEN
		Event.no[3].Text2									:= CONCAT(CONCAT('(',SlavesDiag.FirstErrorSlave.ConfigType), CONCAT(') , ',TO_STRING(NoOfMissedSlaves))) ;
		Event.no[3].pText3									:= ADR(SlavesDiag.FirstErrorSlave.ConfigName);	
	END_IF

	(* Slave State Error *)
	Event.no[4].Flag										:= NoOfSlavesNOK > 0 AND NOT IO.DevStateChanged AND NOT SlavesDiag.Busy AND NOT tonDelTrigDiag.IN;
	IF Event.no[4].Flag
	THEN
		Event.no[4].Text2									:= CONCAT(SlavesDiag.FirstErrorSlave.DevStateText , CONCAT(', Name: ', SlavesDiag.FirstErrorSlave.ConfigName));
		Event.no[4].pText3									:= ADR(SlavesDiag.FirstErrorSlave.ConfigTypeIdentity);	
	END_IF
	
	(* Slave Count Error *)
	Event.no[5].Flag										:= NoOfMissedSlaves <> 0 AND NoOfSlavesNOK > 0 AND NOT ConfirmTrig AND NOT SlavesDiag.Busy AND NOT tonDelTrigDiag.IN;
	IF Event.no[5].Flag
	THEN
		Event.no[5].Text2									:= CONCAT('Cfg Slaves:',CONCAT(TO_STRING(IO.CfgSlaveCount),CONCAT(' | Found:',TO_STRING(IO.SlaveCountTotal))));
		Event.no[5].pText3									:= ADR(SlavesDiag.FirstErrorSlave.ConfigName);
	END_IF	
		
	(* Slaves diag error *)
	Event.no[6].Flag										:= SlavesDiag.Error ;          									
	IF Event.no[6].Flag 									
	THEN    
		Event.no[6].Text2									:= '';            									
		Event.no[6].pText3									:= ADR(SlavesDiag.ErrorText);
	END_IF	
	
	(* Watchdog triggered  *)
	Event.no[7].Flag										:= io.DevStateBits.WatchdogTriggered;	
	IF Event.no[7].Flag 
	THEN 
		Event.no[7].pText3									:= ADR(IO.DevStateText);
	END_IF	
	
	(* DC not in sync  *)
	Event.no[8].Flag										:= IO.DevStateBits.DcNotInSync;
	IF Event.no[8].Flag 
	THEN 
		Event.no[8].pText3									:= ADR(IO.DevStateText);
	END_IF	
	
	(* Out of send ressources  *)
	Event.no[9].Flag										:= IO.DevStateBits.OutOfSendResources;
	IF Event.no[9].Flag 
	THEN 
		Event.no[9].pText3									:= ADR(IO.DevStateText);
	END_IF	

	(* IO locked  *)
	Event.no[10].Flag										:= IO.DevStateBits.IOLockedAfterLinkError;		
	IF Event.no[10].Flag 
	THEN 
		Event.no[10].pText3									:= ADR(IO.DevStateText);
	END_IF
	
	(* Work EventCtrl *)
	Event(
		ConfirmTrig	:= ConfirmTrig,
		SourceId	:= SourceId ,
		no			:= ,
		Disable		:= NOT Enable,
		AutoConfirm := ,
		Status		=> EventStatus);
		
(*****************************************************************************)
END_METHOD

METHOD PUBLIC confirm : bool
VAR_INPUT
END_VAR
confirm			:= Event.confirm();
END_METHOD

END_FUNCTION_BLOCK

// POUs/Fieldbus/Profibus/ProfibusMasterDiag
{attribute 'no_check'}
FUNCTION_BLOCK ProfibusMasterDiag
VAR_INPUT                               					
	Enable													:	BOOL := FALSE;		//FB will be processed as long as enable is TRUE 	
	ResetTrig													:	BOOL := FALSE;		//Resets error with rising edge 
	SourceId												:	UDINT := 103020; 	//default
END_VAR                                 	
VAR_OUTPUT                              	
	IO														:	ProfiBusMasterIO;
END_VAR
VAR
(* trigger ********************************************************)
		
(* events *********************************************************)
	EventMasterError										:	EventHandling;
	EventNoteError											:	ARRAY[1..PARAM.PROFIBUS_MASTER_DEV_IO_MAX_SLAVES] OF EventHandling;
(* function-block *************************************************)
	
(* dummy **********************************************************)	
	i														:	INT;
END_VAR

	(* ProfiBus master diagnosis for EL6731 and slaves	V2.0	*)
	(************************************************************)

(* Work IO ***********************************************)
	IO();

(* Master error ******************************************************)
	EventMasterError(
		Flag			:= IO.Error <> 0 AND Enable,
		ConfirmTrig		:= ResetTrig OR NOT Enable,
		MsgId			:= 1,
		SourceId		:= SourceId,
		eClass			:= ,
		Text1			:= ,
		Text2			:= USINT_TO_STRING(IO.Error),
		pText3			:= ADR(IO.Name),
		State			=> );
		
(* Slave note error **************************************)
	FOR i := IO.MIN_SLAVES TO IO.MAX_SLAVES DO		
		EventNoteError[i](
			Flag		:= IO.SlaveDpStates[i] <> 0 AND Enable,
			ConfirmTrig := ResetTrig OR NOT Enable,
			MsgId		:= TO_UINT(i + 1),
			Text1		:= TO_STRING(i),
			Text2		:= TO_STRING(IO.SlaveDpStates[i]),
			pText3		:= ADR(IO.Name),
			SourceId	:= );
		
 	END_FOR
	

		
(*********************************************************)

END_FUNCTION_BLOCK

// POUs/Fieldbus/Profibus/ProfibusMasterIO
{attribute 'no_check'}
//EL6731 Profibus Master IOs via EtherCAT
FUNCTION_BLOCK ProfibusMasterIO
VAR_OUTPUT CONSTANT
	MIN_SLAVES												:	INT := 1;
	MAX_SLAVES												:	INT := PARAM.PROFIBUS_MASTER_DEV_IO_MAX_SLAVES;
END_VAR
VAR_INPUT
END_VAR
VAR_OUTPUT
	DevId											AT %I*	: 	UINT; 		//// Link to Profibus "DevId" or EtherCAT Master "DevId" under InfoData 
	AdsAddr											AT %I*	:	AMSADDR;	//Structure of AdsAddr
	AmsNetIdStr												:	T_AmsNetId;	//shows string of AmsNetId 
	Error											AT %I*	:	USINT;		//No of Slaves with an state <> 0
	ActualModulo		 							AT %I*	:	USINT;		
	DiagFlag										AT %I*	:	BOOL;		//TRUE when diagnostic values are available
	Name													:	STRING(30);
                            					             	
	SlaveDpStates									AT %I*	:	ARRAY[MIN_SLAVES..MAX_SLAVES] OF USINT;
	SlaveExtDiagFlags								AT %I*	:	ARRAY[MIN_SLAVES..MAX_SLAVES] OF BOOL;
END_VAR                     					             	
VAR                         	                             	
	IOF_GetBoxNameByAddr									:	IOF_GetBoxNameByAddr := (NETID := '', TMOUT := DEFAULT_ADS_TIMEOUT);
END_VAR

(* Profibus Master IO diag										      	 		*)
(********************************************************************************)

(* Get name ******************************************************************************)
IF Name = ''
	AND AdsAddr.port <> 0 AND DevId <> 0
	OR IOF_GetBoxNameByAddr.BUSY
	OR IOF_GetBoxNameByAddr.START
THEN
	AmsNetIdStr												:= F_CreateAmsNetId(nIds := AdsAddr.netId);

	IF AmsNetIdStr = '0.0.0.0.0.0' THEN
		AmsNetIdStr	:= '';
	END_IF
		
	IOF_GetBoxNameByAddr(
		NETID		:= AmsNetIdStr , 
		DEVICEID	:= UINT_TO_UDINT(DevId) ,
		BOXADDR		:= AdsAddr.port ,
		START		:= Name = '' AND NOT IOF_GetBoxNameByAddr.BUSY,
		TMOUT		:= ,
		BOXNAME		=> name);
END_IF
(********************************************************************************)

END_FUNCTION_BLOCK

// POUs/Fieldbus/Profinet/ProfinetControllerIO
{attribute 'no_check'}
//EL6631 Profinet Controller IOs via EtherCAT
FUNCTION_BLOCK ProfinetControllerIO EXTENDS EcSlaveInfoDataExt
VAR_OUTPUT CONSTANT
	MIN_BOX													:	INT := 1;
	MAX_BOX													:	INT := PARAM.PROFINET_CONTROLLER_DEV_IO_MAX_BOX;
END_VAR
VAR_INPUT
	DevCtrl			 								AT %Q*	:	UINT;
	PnIoBoxCtrl										AT %Q*	:	ARRAY[MIN_BOX ..MAX_BOX] OF UINT;
END_VAR
VAR_OUTPUT
//Device parameter
	DevState		 								AT %I*	:	UINT;		//Link to master device state
	PnIoError										AT %I*	:	UINT;		//Link to master IO error
	PnIoDiag										AT %I*	:	UINT;		//Link to master IO Diag 
                         				
	AoeNetId										AT %I*	:	AMSNETID;		//Link to master AoeNetID
//Box states	             	
	PnIoBoxState									AT %I*	:	ARRAY[MIN_BOX ..MAX_BOX] OF UINT; //Link to box state
	PnIoBoxDiag										AT %I*	:	ARRAY[MIN_BOX ..MAX_BOX] OF UINT; //Link to box diag	
END_VAR                     					             	
VAR       
END_VAR

SUPER^();

END_FUNCTION_BLOCK

// POUs/IO/_EcSlaveInfoDataIO/EcSlaveInfoDataExt
{attribute 'no_check'}
{attribute 'reflection'} 
FUNCTION_BLOCK EcSlaveInfoDataExt Extends EcSlaveInfoData
VAR_INPUT
END_VAR                         					
VAR_OUTPUT                      					
	AmsNetIdStr												: T_AmsNetId; //AMS NetID string
	EcMasterDevId									AT %I*	: UINT; 	// Link to EtherCAT Master "DevId" under InfoData 
	DevName													:	STRING(30) := ''; //Slave device name as give in IO tree				
	{attribute 'instance-path'} 
    {attribute 'noinit'} 
    InstancePath 											: STRING; 	
END_VAR
VAR
	IOF_GetBoxNameByAddr									:	IOF_GetBoxNameByAddr := (NETID := '', TMOUT := DEFAULT_ADS_TIMEOUT);
	_Init_													: BOOL;
END_VAR

(* Get device name by address and master device id								*)
(********************************************************************************)

(* Get name *********************************************************************)
IF NOT _Init_
THEN 	
	IF NOT IOF_GetBoxNameByAddr.START
	THEN
		IF AdsAddr.port = 0 
		THEN
			adsLogError('AdsAddr.port invalid: %s', InstancePath);
		END_IF
		IF EcMasterDevId = 0 
		THEN
			adsLogError('EcMasterDevId invalid: %s', InstancePath);
		END_IF
			
		IF AdsAddr.port > 0 AND EcMasterDevId > 0
		THEN
			IOF_GetBoxNameByAddr.START						:= TRUE;
			AmsNetIdStr										:= F_CreateAmsNetId(nIds := AdsAddr.netId);
		END_IF		
	END_IF
	
	IOF_GetBoxNameByAddr(
		NETID		:=  , (* Local *)
		DEVICEID	:= TO_UDINT(EcMasterDevId) ,
		BOXADDR		:= AdsAddr.port ,
		START		:= ,
		TMOUT		:= ,
		BOXNAME		=> DevName);
	IF NOT IOF_GetBoxNameByAddr.BUSY 
	THEN
		IF IOF_GetBoxNameByAddr.ERR 
		THEN
			adsLogError(CONCAT(CONCAT('ADS Error ', DWORD_TO_HEXSTR(IOF_GetBoxNameByAddr.ERRID,4,FALSE)),' reading BoxName of EtherCAT Device: %s'), InstancePath);
		END_IF
		IOF_GetBoxNameByAddr(START:= FALSE);
		_Init_												:= TRUE;
	END_IF
END_IF
(********************************************************************************)

END_FUNCTION_BLOCK

// POUs/IO/_EcSlaveInfoDataIO/EcSlaveInfoData
{attribute 'no_check'}
FUNCTION_BLOCK EcSlaveInfoData implements I_EcSlaveInfoData
VAR_INPUT
END_VAR
VAR_OUTPUT
	WcState											AT  %I*		:	BOOL;			//TRUE=Invalid - TRUE an invalid working counter and FALSE a valid working counter 
	InputToggle										AT  %I*		:	BOOL;			//variable toggles in every successful cycle	
	{attribute 'displaymode':='hex'}  
	InfoDataState									AT  %I*		: 	UINT;			(* current EtherCAT device state:
																						EC_DEVICE_STATE_MASK		:BYTE 	:=16#0F;
																						EC_DEVICE_STATE_INIT		:BYTE 	:=16#01;
																						EC_DEVICE_STATE_PREOP		:BYTE 	:=16#02;
																						EC_DEVICE_STATE_BOOTSTRAP	:BYTE 	:=16#03;
																						EC_DEVICE_STATE_SAFEOP		:BYTE 	:=16#04;
																						EC_DEVICE_STATE_OP			:BYTE 	:=16#08;
																						EC_DEVICE_STATE_ERROR		:BYTE 	:=16#10;
																						EC_DEVICE_STATE_INVALID_VPRS :BYTE 	:=16#20;
																						EC_DEVICE_STATE_INITCMD_ERROR:BYTE 	:=16#40; *)
	AdsAddr											AT  %I*		:	AMSADDR; 		//Slave device AdsAddr structure(ID and port number)
END_VAR
VAR
END_VAR

;

PROPERTY PUBLIC rInfoData : reference to EcSlaveInfoData
GET
rInfoData := THis^;
END_GET
END_PROPERTY

END_FUNCTION_BLOCK

// POUs/IO/_EcSlaveInfoDataIO/I_EcSlaveInfoData
INTERFACE I_EcSlaveInfoData EXTENDS __SYSTEM.IQueryInterface

PROPERTY PUBLIC rInfoData : reference to EcSlaveInfoData
GET
END_GET
END_PROPERTY

END_INTERFACE

// POUs/Fieldbus/Profinet/ProfinetControllerIO_wEvents
{attribute 'no_check'}
//EL6631 Profinet Controller IOs via EtherCAT
FUNCTION_BLOCK ProfinetControllerIO_wEvents EXTENDS ProfinetControllerIO
VAR_OUTPUT CONSTANT

END_VAR
VAR_INPUT
	Enable													:	BOOL := FALSE;
	ResetTrig												:	BOOL := FALSE;
	SourceId												:	UDINT := 103040; (* default *)	
END_VAR
VAR_OUTPUT

END_VAR                     					             	
VAR   
(* trigger ********************************************************)
	
(* events *********************************************************)
	EventControllerError									:	EventHandling;
	EventBoxError											:	ARRAY[1..MAX_BOX] OF EventHandling;
	
(* function-block *************************************************)
	
(* dummy **********************************************************)	
	i														:	INT;    
END_VAR

	(* Profinet controller diagnosis for EL6631	and boxes	V3.0*)
	(************************************************************)

(* Work super ***********************************************)
SUPER^();
	
(* Master error *******************************************)
	EventControllerError(
		Flag				:= PnIoError <> 0 AND Enable,
		ConfirmTrig			:= ResetTrig OR NOT Enable,
		MsgId				:= 1,
		SourceId			:= SourceId,
		eClass				:= ,
		Text1				:= TO_STRING(PnIoError),
		Text2				:= ,
		pText3				:= ADR(DevName),
		State				=> );

(* Box error *********************************************)
	FOR i := MIN_BOX TO MAX_BOX DO
		EventBoxError[i](
			Flag			:= PnIoBoxDiag[i] <> 0 AND Enable,
			ConfirmTrig		:= ResetTrig OR NOT Enable,
			MsgId			:= TO_UINT(i + 1),
			SourceId		:= SourceId,
			eClass			:= ,
			Text1			:= TO_STRING(PnIoBoxDiag[i]),
			Text2			:= TO_STRING(i),
			pText3			:= ADR(DevName),
			State			=> );
 	END_FOR

(*********************************************************)

END_FUNCTION_BLOCK

// POUs/Fieldbus/Profinet/ProfinetDeviceIO
{attribute 'no_check'}
//EL6631-0010 Profinet Device IOs via EtherCAT
// it´s possible to set up multi device for diffrent master
FUNCTION_BLOCK ProfinetDeviceIO EXTENDS EcSlaveInfoDataExt
VAR_OUTPUT CONSTANT
	MIN_BOX													:	INT := 1;
	MAX_BOX													:	INT := PARAM.PROFINET_DEVICE_DEV_IO_MAX_BOX;
																
END_VAR
VAR_INPUT
	PnIoBoxCtrl										AT %Q*	:	ARRAY[MIN_BOX ..MAX_BOX] OF UINT;
END_VAR
VAR_OUTPUT                       				
	AoeNetId										AT %I*	:	AMSNETID;		//Link to master AoeNetID
//Box states	             	
	{attribute 'displaymode':='binary'}
	PnIoBoxState									AT %I*	:	ARRAY[MIN_BOX ..MAX_BOX] OF UINT; //Link to box state
END_VAR                     					             	
VAR       
END_VAR

SUPER^();

END_FUNCTION_BLOCK

// POUs/FileHandling/Basic/FileHandling
{attribute 'no_check'}
//Wrapper for all file fucntions provided by lib Tc2_TcSystem.Lib, see Beckhoff information system for detailed information of each function. 
FUNCTION_BLOCK FileHandling EXTENDS FbBase
VAR_OUTPUT CONSTANT
	FNC_OPEN												:	INT := 0; //With this function a new file can be created, or a closed existing file can be re-opened for further processing
	FNC_READ												:	INT := 1; //With this function  the contents of an already opened file can be read. The file must have been already opened for read access
	FNC_WRITE												:	INT := 2; //Data can be written into a file with this function if it is opened in write mode
	FNC_PUTS												:	INT := 3; //The function writes strings to the file if it is opened in write mode
	FNC_GETS												:	INT := 4; //The function reads zero terminated strings from a file and moves the file pointer to the next line.(if pBuffer is <> 0, the read line will copied to the buffer as well)
	FNC_CLOSE												:	INT := 5; //With this function the file can be closed, and thereby placed into a defined state for further processing by other programs
	FNC_DELETE												:	INT := 6; //With this function the existing file can be deleted
	FNC_RENAME												:	INT := 7; //With this function the existing file can be renamed.
	FNC_REMOVEDIR											:	INT := 8; //This function removes a directory from the data medium. A directory containing data can not be removed!
	FNC_CREATEDIR											:	INT := 9; //This function creates new directories on the data medium.
	FNC_SEEK												:	INT := 10;//With this function the file pointer of an opened file can be set to a definable position
	FNC_TELL												:	INT := 11;//The function gets the current position of the file pointer. The position is expressed as an offset relative to the beginning of the stream.
	FNC_EOF													:	INT := 12;//The function tests for the end-of-file.
	FNC_LOAD												:	INT := 13;//The file is opened implicitly in binary mode, the contents are read out and the file is then closed again.
END_VAR             										                 										
VAR_INPUT           										
	Fnc														:	INT (FNC_OPEN..FNC_LOAD) := FNC_OPEN; //Parameter for requested function
	AMSNetId												:	T_AmsNetId := ''; //Ams Net Id 
	Timeout													:	TIME := DEFAULT_ADS_TIMEOUT; //Ads timeout 
	Mode													:	DWORD := FOPEN_MODEAPPEND OR FOPEN_MODEPLUS OR FOPEN_MODETEXT; 
																			(* 	FOPEN_MODEREAD "r": Opens for reading. If the file does not exist or cannot be found, the call fails.
																				FOPEN_MODEWRITE  "w": Opens an empty file for writing. If the given file exists, its contents are destroyed.
																				FOPEN_MODEAPPEND  "a": Opens for writing at the end of the file (appending) without removing the EOF marker before writing new data to the file; creates the file first if it doesn’t exist.
																				FOPEN_MODEREAD OR FOPEN_MODEPLUS  "r+": Opens for reading and writing. The file must exist.
																				FOPEN_MODEWRITE OR FOPEN_MODEPLUS  "w+": Opens an empty file for both reading and writing. If the given file exists, its contents are destroyed.
																				FOPEN_MODEAPPEND OR FOPEN_MODEPLUS  "a+": 	Opens for reading and appending; the appending operation includes the removal of the EOF marker before new data is written to the file and the EOF marker is restored after writing is complete; creates the file first if it doesn’t exist.
																															When a file is opened with the "a" or "a+" access type, all write operations occur at the end of the file. The file pointer can be repositioned using FB_FileSeek, but is always moved back to the end of the file before any write operation is carried out. Thus, existing data cannot be overwritten. 																				                                    								
																				FOPEN_MODEBINARY  "b": Open in binary (untranslated) mode.
																				FOPEN_MODETEXT  "t": Open in text (translated) mode. *)
	Path													:	T_MaxString; // \\PC-Name\Folder\ 
	FileName												:	T_MaxString := ''; // NewFile.xyz 
	OldFileName												:	T_MaxString := ''; // File.xyz 
	pBuffer													:	PVOID; //pointer to data section 
	Length													: 	UDINT; // sizeof data section for read and write. Note to use "LEN" while writing-command, beacause otherwise the whole datasection and not only the string will be written 
	SeekOrigin												: 	E_SeekOrigin := SEEK_SET; //Seek function parameter - Contains the relative position for the move.
	SeekPos													:	DINT; //Seek function parameter - Contains the desired (new) target position of the file pointer.
END_VAR
VAR_OUTPUT
	EOF														:	BOOL;	//This output is switched to TRUE if the end of file is reached.
	WorkedLen												:	UDINT;	//Contains the number of bytes currently read or written
	hFile													:	UINT;	//File handle of currently opened file
	ActSeekPos												:	DINT;	//Act file pointer position of filled by Tell function
	Line   													: T_MaxString; //Read line of file - filled by function Gets

END_VAR
VAR
(* internal used variables ************************************************************)
	MemErrorText											:	STRING(50);
	MemFnc													:	INT := -1;
	
(* trigger ******************************************************************************)

(* function-block instances ************************************************************)
	File_Open												:	FB_FileOpen;
	File_Close												: 	FB_FileClose;
	File_Read 												: 	FB_FileRead;
	File_Write												:	FB_FileWrite;
	File_Delete												:	FB_FileDelete;
	File_Rename												:	FB_FileRename;
	File_Puts												:	FB_FilePuts;
	File_Gets												:	FB_FileGets;
	File_CreateDir											:	FB_CreateDir;
	File_RemoveDir											:	FB_RemoveDir;
	File_Tell												:	FB_FileTell ;
	File_Seek												:	FB_FileSeek ;
	File_EoF												:	FB_EOF;
	File_Load												:	FB_FileLoad;
END_VAR

	(* FileHandling												V2.0	*)
	(********************************************************************)

(* Sequence **********************************************************************)
	rtExecute(CLK := Execute);
	IF rtExecute.Q
		AND MemFnc < 0
	THEN
		Busy												:= TRUE;
		Done												:= FALSE;
		Error												:= FALSE;
		ErrorId												:= 0;
		CASE fnc OF                     					
		FNC_OPEN:		MemFnc 								:= fnc;
		FNC_READ:		MemFnc 								:= fnc;
		FNC_WRITE:		MemFnc 								:= fnc;
		FNC_PUTS:		MemFnc 								:= fnc;
		FNC_GETS:		MemFnc 								:= fnc;
		FNC_CLOSE:		MemFnc 								:= fnc;
		FNC_DELETE:		MemFnc 								:= fnc;
		FNC_RENAME:		MemFnc 								:= fnc;
		FNC_REMOVEDIR: 	MemFnc 								:= fnc;
		FNC_CREATEDIR: 	MemFnc 								:= fnc;
		FNC_SEEK:		MemFnc 								:= fnc;
		FNC_TELL:		MemFnc 								:= fnc;
		FNC_EOF:		MemFnc 								:= fnc;
		FNC_LOAD:		MemFnc 								:= fnc;
		ELSE                            					
			ErrorId											:= E_AdsErr.DEVICE_INVALIDPARM;
			Error											:= TRUE;
			Done											:= FALSE;
			Busy											:= FALSE;
		END_CASE
	END_IF

	CASE MemFnc OF
		FNC_OPEN:		Open(Execute := Execute);
		FNC_READ:		Read(Execute := Execute);
		FNC_WRITE:		Write(Execute := Execute);
		FNC_PUTS:		Puts(Execute := Execute);
		FNC_GETS:		Gets(Execute := Execute);
		FNC_CLOSE:		Close(Execute := Execute);
		FNC_DELETE:		Delete(Execute := Execute);
		FNC_RENAME:		Rename(Execute := Execute);
		FNC_REMOVEDIR: 	RemoveDir(Execute := Execute);
		FNC_CREATEDIR: 	CreateDir(Execute := Execute);
		FNC_SEEK:		Seek(Execute := Execute);
		FNC_TELL:		Tell(Execute := Execute);
		FNC_EOF:		IsEof(Execute := Execute);
		FNC_LOAD:		Load(Execute := Execute);
	
	-1:
		IF NOT Execute
		THEN
			Busy											:= FALSE;
			Done											:= FALSE;
			Error											:= FALSE;
			ErrorID											:= 0;
		END_IF
	END_CASE
(*************************************************************************)

METHOD PUBLIC close : Bool //Return value = TRUE if busy
VAR_INPUT
	Execute		:	BOOL	:= FALSE;
END_VAR
	IF Execute
	THEN
		Error												:=	FALSE;
		ErrorId												:= 0;
		File_Close.bExecute 								:= TRUE;
	ELSIF NOT File_Close.bBusy      						
	THEN                            						
		Error												:=	FALSE;
		ErrorId												:= 0;
		File_Close.bExecute 								:= FALSE;
	END_IF                          						
                                    	
	MemFnc 													:= FNC_CLOSE;
	THIS^.Execute											:= Execute;

	File_Close(
		sNetId		:= AMSNetId,
		hFile		:= hFile,
		bExecute	:= ,
		tTimeout	:= Timeout,
		bBusy		=> Busy,
		bError		=> ,
		nErrId		=> );

	IF NOT File_Close.bBusy
		AND NOT File_Close.bError
		AND File_Close.bExecute
	THEN
		Done												:= TRUE;
		hFile 												:= 0;
	ELSE                            						
		Done												:= FALSE;
	END_IF

	IF NOT Busy
	THEN
		IF File_Close.bExecute
		THEN
			Error											:=	File_Close.bError;
			ErrorId											:= File_Close.nErrId;
		END_IF
		IF NOT Execute
		THEN
			MemFnc											:=  -1;
			File_Close(bExecute 							:= FALSE);
		END_IF
	END_IF

	(* Fehler speichern *)
	IF Error
	THEN
		MemErrorText										:= CONCAT('File_Close ErrorID: ', UDINT_TO_STRING(ErrorID));
	END_IF
	
	Close													:= Busy;
END_METHOD

METHOD PUBLIC createDir : BOOL //Return value = TRUE if busy
//required parameter
//Path
VAR_INPUT
	Execute													:	BOOL;
END_VAR
	IF Execute
	THEN
		Error												:=	FALSE;
		ErrorId												:= 0;
		File_CreateDir.bExecute 							:= TRUE;
	ELSIF NOT File_CreateDir.bBusy      					
	THEN                                					
		Error												:=	FALSE;
		ErrorId												:= 0;
		File_CreateDir.bExecute								:= FALSE;
	END_IF                              					
                                        	
	MemFnc 													:= FNC_CREATEDIR;
	THIS^.Execute											:= Execute;

	File_CreateDir(
		sNetId		:= AMSNetId,
		sPathName	:= Path,
		ePath		:= ,
		bExecute	:= ,
		tTimeout	:= Timeout,
		bBusy		=> Busy,
		bError		=> ,
		nErrId		=> );

	Done													:= NOT File_CreateDir.bBusy
																AND NOT File_CreateDir.bError
																AND File_CreateDir.bExecute;
	IF NOT Busy
	THEN
		IF File_CreateDir.bExecute
		THEN
			Error											:=	File_CreateDir.bError;
			ErrorId											:= File_CreateDir.nErrId;
		END_IF
		IF NOT Execute
		THEN
			MemFnc											:=  -1;
			File_CreateDir(bExecute := FALSE);
		END_IF
	END_IF


	IF Error
	THEN
		MemErrorText										:= CONCAT('File_CreateDir ErrorID: ', UDINT_TO_STRING(ErrorID));
	END_IF
	
	CreateDir												:= Busy;
END_METHOD

METHOD PUBLIC delete : BOOL //Return value = TRUE if busy
//required parameter
//Path
//FileName
VAR_INPUT
	Execute			:	bool;
END_VAR
	IF Execute
	THEN
		Error												:=	FALSE;
		ErrorId												:= 0;
		File_Delete.bExecute 								:= TRUE;
	ELSIF NOT File_Delete.bBusy         					
	THEN                                					
		Error												:=	FALSE;
		ErrorId												:= 0;
		File_Delete.bExecute 								:= FALSE;
	END_IF                              					
                                        	
	MemFnc 													:= FNC_DELETE;
	THIS^.Execute											:= Execute;

	File_Delete(
		sNetId		:= AMSNetId,
		sPathName	:= CONCAT(Path,FileName),
		ePath		:= ,
		bExecute	:= ,
		tTimeout	:= Timeout,
		bBusy		=> Busy,
		bError		=> ,
		nErrId		=> );

	Done													:= 	NOT File_Delete.bBusy
																AND NOT File_Delete.bError
																AND File_Delete.bExecute;
	IF NOT Busy
	THEN
		IF File_Delete.bExecute
		THEN
			Error											:=	File_Delete.bError;
			ErrorId											:= File_Delete.nErrId;
		END_IF
		IF NOT Execute
		THEN
			MemFnc											:= -1;
			File_Delete(bExecute := FALSE);
		END_IF
	END_IF


	IF Error
	THEN
		MemErrorText										:= CONCAT('File_Delete ErrorID: ', UDINT_TO_STRING(ErrorID));
	End_if
	
	Delete													:= Busy;
END_METHOD

METHOD PUBLIC gets : BOOL //Return value = TRUE if busy
//required parameter
//Path
//Filename
//Mode
//pBuffer
VAR_INPUT
	Execute			:	BOOL;
END_VAR
IF pBuffer = 0 THEN
	Busy													:= NOT Error;
	Error													:= TRUE;
	ErrorId													:= E_AdsErr.DEVICE_INVALIDPARM;
	Done													:= FALSE;
	MemFnc													:= -1 ;
	RETURN;                             					
END_IF                                  					
                                        					
	MemFnc 													:= FNC_GETS;
	THIS^.Execute											:= Execute;
                                        					
	CASE State OF                       	
	0:                                  	
		IF Execute                      	
		THEN                            	
			Done											:= FALSE;
			Error											:= FALSE;
			ErrorId 										:= 0;
			
			File_Open(bExecute := FALSE);
			File_Gets(bExecute := FALSE);
			File_Close(bExecute := FALSE);
			
			EOF												:= FALSE;
			WorkedLen										:= 0;
			
			IF hFile = 0
			THEN
				File_Open(
					sNetId		:= AMSNetId,
					sPathName	:= CONCAT(Path,FileName),
					nMode		:= Mode ,
					ePath		:= (* Default *),
					bExecute	:= TRUE,
					tTimeout	:= Timeout,
					bBusy		=> ,
					bError		=> ,
					nErrId		=> ,
					hFile		=> );

				State 										:= 10;
			ELSE                							
				State 										:= 10;
			END_IF
		ELSE
			Done											:= FALSE;
			Error											:= FALSE;
			ErrorId 										:= 0;
		END_IF

	10:
		File_Open();

		IF NOT File_Open.bBusy
		THEN
			IF File_Open.bError
			THEN
				State 										:= 99;
			ELSE
				IF File_Open.bExecute THEN hFile := File_Open.hFile; END_IF
				File_Gets(
					sNetId		:= AMSNetId,
					hFile		:= hFile,
					bExecute	:= TRUE,
					tTimeout	:= Timeout,
					sLine		=> ,
					bEOF		=> ,
					bBusy		=> ,
					bError		=> ,
					nErrId		=> );

				State 										:= 20;
			END_IF
		END_IF

	20:
		File_Gets(bEOF		=> EOF);
		IF NOT File_Gets.bBusy
		THEN
			IF NOT File_Gets.bError
			THEN
				IF pBuffer <> 0 AND Length <> 0
				THEN
					 MEMCPY(pBuffer , ADR(File_Gets.sLine), MIN(TO_UDINT(Length), SIZEOF(File_Gets.sLine)));
				END_IF
				Line										:= File_Gets.sLine;
			END_IF
			IF File_Open.bExecute
			THEN
				File_Close(
					sNetId	:= AMSNetId,
					hFile	:= hFile,
					bExecute:= TRUE,
					tTimeout:= Timeout,
					bBusy	=> ,
					bError	=> ,
					nErrId	=> );
				State										:= 30;
			ELSE
				State										:= 99;
			END_IF

		END_IF

	30:
		File_Close();
		IF NOT File_Close.bBusy
		THEN
			hFile											:= 0;
			State											:= 99;
		END_IF

	99:
		IF NOT Execute
		THEN
			Memfnc											:= -1;
			state 											:= 0;
		END_IF
	END_CASE

	Done													:= state = 99
																AND NOT File_Gets.bError
																AND NOT File_Close.bError
																AND NOT File_Open.bError;
                                        					
	Error													:= state = 99
																AND(
																File_Gets.bError
																OR File_Close.bError
																OR File_Open.bError);
                                        					
	Busy													:= state <> 0
																AND NOT Done
																AND NOT Error;

	IF Error
	THEN
		IF File_Close.bError 	THEN 	ErrorId :=  File_Close.nErrId; 	END_IF
		IF File_Gets.bError 	THEN 	ErrorId :=  File_Gets.nErrId; 	END_IF
		IF File_Open.bError 	THEN	ErrorId :=  File_Open.nErrId; 	END_IF
	ELSE
		ErrorId 											:= 0;
	END_IF                              					
                                        					
	IF NOT Execute                      					
		AND state = 99                  					
	THEN                                					
			MemFnc											:= -1;
		state 												:= 0;
	END_IF                              	
                                        	
	IF Error                            	
	THEN                                	
		MemErrorText										:= CONCAT('File_Gets ErrorID: ', UDINT_TO_STRING(ErrorID));
	END_IF                              					
                                        					
	Gets													:= Busy;
END_METHOD

METHOD PUBLIC isEoF : BOOL //Return value = TRUE if busy
VAR_INPUT
	Execute													:	BOOL;
END_VAR
	IF Execute
	THEN
		Error												:=	FALSE;
		ErrorId												:= 0;
		File_EoF.bExecute 									:= TRUE;
	ELSIF NOT File_EoF.bBusy           					
	THEN                                					
		Error												:=	FALSE;
		ErrorId												:= 0;
		File_EoF.bExecute 									:= FALSE;
	END_IF                              							
	                                    	
	MemFnc 													:= FNC_EOF;
	THIS^.Execute											:= Execute;
                                        	
	File_EoF(
		sNetId		:= AMSNetId,
		hFile		:= hFile ,
		tTimeout	:= Timeout,
		bBusy		=> Busy,
		bError		=> ,
		nErrId		=> ,
		bEoF		=> EoF);

	Done													:= NOT File_EoF.bBusy
																AND NOT File_EoF.bError
																AND File_EoF.bExecute;
	IF NOT Busy                         					
	THEN                        					
		IF File_EoF.bExecute           					
		THEN                            	
			Error											:=	File_EoF.bError;
			ErrorId											:= File_EoF.nErrId;
		END_IF
		IF NOT Execute
		THEN
			MemFnc											:= 1;
			File_EoF(bExecute := FALSE);
		END_IF
	END_IF


	IF Error
	THEN
		MemErrorText										:= CONCAT('File_EoF ErrorID: ', UDINT_TO_STRING(ErrorID));
	END_IF
	
	IsEoF													:= Busy;
END_METHOD

METHOD PUBLIC load : BOOL //Result = Busy
//required parameter
//Path
//FileName
VAR_INPUT
	Execute				:	BOOL; 
END_VAR
IF Execute
THEN
	Error													:= FALSE;
	ErrorId													:= 0;
	File_Load.bExecute 										:= TRUE;
ELSIF NOT File_Load.bBusy           						
THEN                                						
	Error													:=	FALSE;
	ErrorId													:= 0;
	File_Load.bExecute 										:= FALSE;
END_IF	

MemFnc 														:= FNC_LOAD;
THIS^.Execute												:= Execute;

(* Work File Load *)
File_Load(
	sNetId		:= AMSNetId, 
	sPathName	:= CONCAT(Path,FileName), 
	pReadBuff	:= pBuffer, 
	cbReadLen	:= Length, 
	bExecute	:= , 
	tTimeout	:= Timeout, 
	bBusy		=> Busy, 
	bError		=> , 
	nErrId		=> , 
	cbRead		=> WorkedLen);
Done														:= NOT File_Load.bBusy
																AND NOT File_Load.bError
																AND File_Load.bExecute;
IF NOT Busy
THEN
	IF File_Load.bExecute
	THEN
		Error												:= File_Load.bError;
		ErrorId												:= File_Load.nErrId;
	END_IF
	IF NOT Execute
	THEN
		MemFnc												:= -1;
		File_Load(bExecute := FALSE);
	END_IF
END_IF

IF Error
THEN
	MemErrorText											:= CONCAT('File_Load ErrorID: ', UDINT_TO_STRING(ErrorID));
END_IF                              						
                                    	
load														:= Busy;
END_METHOD

METHOD PUBLIC open : BOOL //Return value = TRUE if busy
//required parameter
//Path
//FileName
//Mode
VAR_INPUT
	Execute				:	BOOL; 
END_VAR
IF Execute
THEN
	Error													:= FALSE;
	ErrorId													:= 0;
	File_Open.bExecute 										:= TRUE;
ELSIF NOT File_Open.bBusy           						
THEN                                						
	Error													:=	FALSE;
	ErrorId													:= 0;
	File_Open.bExecute 										:= FALSE;
END_IF	

MemFnc 														:= FNC_OPEN;
THIS^.Execute												:= Execute;

(* Work File Open *)
File_Open(
	sNetId		:= AMSNetId,
	sPathName	:= CONCAT(Path,FileName),
	nMode		:= Mode ,
	ePath		:= (* Default *),
	bExecute	:= ,
	tTimeout	:= Timeout,
	bBusy		=> Busy,
	bError		=> ,
	nErrId		=> ,
	hFile		=> hFile);

Done														:= NOT File_Open.bBusy
																AND NOT File_Open.bError
																AND File_Open.bExecute;
IF NOT Busy
THEN
	IF File_Open.bExecute
	THEN
		Error												:=	File_Open.bError;
		ErrorId												:= File_Open.nErrId;
	END_IF
	IF NOT Execute
	THEN
		MemFnc												:= -1;
		File_Open(bExecute := FALSE);
	END_IF
END_IF

IF Error
THEN
	MemErrorText											:= CONCAT('File_Open ErrorID: ', UDINT_TO_STRING(ErrorID));
END_IF                              						
                                    	
Open														:= Busy;
END_METHOD

METHOD PUBLIC puts : BOOL //Return value = TRUE if busy
//required parameter
//Path
//FileName
//Mode
//pBuffer
//Lenght
VAR_INPUT
	Execute				:	BOOL;
END_VAR
IF pBuffer = 0 THEN
	Busy													:= NOT Error;
	Error													:= TRUE;
	ErrorId													:= E_AdsErr.DEVICE_INVALIDPARM;
	Done													:= FALSE;
	MemFnc													:= -1 ;
	RETURN;
END_IF

	MemFnc 													:= FNC_PUTS;
	THIS^.Execute											:= Execute;

	CASE State OF
	0:
		IF Execute
		THEN
			Done											:= FALSE;
			Error											:= FALSE;
			ErrorId 										:= 0;
			
			File_Open(bExecute := FALSE);
			File_Puts(bExecute := FALSE);
			File_Close(bExecute := FALSE);
			
			EOF												:= FALSE;
			WorkedLen										:= 0;
			
			IF hFile = 0
			THEN
				File_Open(
					sNetId		:= AMSNetId,
					sPathName	:= CONCAT(Path,FileName),
					nMode		:= Mode ,
					ePath		:= (* Default *),
					bExecute	:= TRUE,
					tTimeout	:= Timeout,
					bBusy		=> ,
					bError		=> ,
					nErrId		=> ,
					hFile		=> );

				State 										:= 10;
			ELSE                							
				State 										:= 10;
			END_IF              							
		ELSE                    							
			Done											:= FALSE;
			Error											:= FALSE;
			ErrorId 										:= 0;
		END_IF

	10:
		File_Open();

		IF NOT File_Open.bBusy
		THEN
			IF File_Open.bError
			THEN
				State 										:= 99;
			ELSE
				IF File_Open.bExecute THEN hFile := File_Open.hFile; END_IF
				MEMCPY(ADR(File_Puts.sLine),  pBuffer, MIN(TO_UDINT(Length), SIZEOF(File_Puts.sLine)));
				File_Puts(
					sNetId		:= AMSNetId,
					hFile		:= hFile,
					sLine		:= (* siehe oben *),
					bExecute	:= TRUE,
					tTimeout	:= Timeout,
					bBusy		=> ,
					bError		=> ,
					nErrId		=> );

				State 										:= 20;
			END_IF
		END_IF

	20:
		MEMCPY(ADR(File_Puts.sLine),  pBuffer, MIN(TO_UDINT(Length), SIZEOF(File_Puts.sLine)));
		File_Puts();

		IF NOT File_Puts.bBusy
		THEN
			IF File_Open.bExecute
			THEN
				File_Close(
					sNetId	:= AMSNetId,
					hFile	:= hFile,
					bExecute:= TRUE,
					tTimeout:= Timeout,
					bBusy	=> ,
					bError	=> ,
					nErrId	=> );
				State										:= 30;
			ELSE
				State										:= 99;
			END_IF

		END_IF

	30:
		File_Close();
		IF NOT File_Close.bBusy
		THEN
			hFile						:= 0;
			State						:= 99;
		END_IF

	99:
		IF NOT Execute
		THEN
			Memfnc					:= -1;
			state 					:= 0;
		END_IF
	END_CASE

	Done							:= state = 99
										AND NOT File_Puts.bError
										AND NOT File_Close.bError
										AND NOT File_Open.bError;

	Error							:= state = 99
										AND(
										File_Puts.bError
										OR File_Close.bError
										OR File_Open.bError);

	Busy							:= state <> 0
										AND NOT Done
										AND NOT Error;

	IF Error
	THEN
		IF File_Close.bError 	THEN	ErrorId :=  File_Close.nErrId; 	END_IF
		IF File_Puts.bError 	THEN 	ErrorId :=  File_Puts.nErrId; 	END_IF
		IF File_Open.bError 	THEN 	ErrorId :=  File_Open.nErrId;	END_IF
	ELSE
		ErrorId 					:= 0;
	END_IF

	IF NOT Execute
		AND state = 99
	THEN
		MemFnc						:= -1;
		state 						:= 0;
	END_IF

	IF Error
	THEN
		MemErrorText				:= CONCAT('File_Puts ErrorID: ', UDINT_TO_STRING(ErrorID));
	END_IF
	
	Puts							:= Busy;
END_METHOD

METHOD PUBLIC read : BOOL //Return value = TRUE if busy
//required parameter
//Path
//FileName
//Mode
//pBuffer
//Lenght
VAR_INPUT
	Execute			:	BOOL;
END_VAR
IF pBuffer = 0 THEN
	Busy													:= NOT Error;
	Error													:= TRUE;
	ErrorId													:= E_AdsErr.DEVICE_INVALIDPARM;
	Done													:= FALSE;
	MemFnc													:= -1 ;
	RETURN;                             					
END_IF                                  					
                                        	
	MemFnc 													:= FNC_READ;
	THIS^.Execute											:= Execute;

	CASE State OF
	0:
		IF Execute
		THEN
			Done											:= FALSE;
			Error											:= FALSE;
			ErrorId 										:= 0;
			
			File_Open(bExecute := FALSE);
			File_Read(bExecute := FALSE);
			File_Close(bExecute := FALSE);
			
			EOF												:= FALSE;
			WorkedLen										:= 0;
			
			IF hFile = 0
			THEN
				File_Open(
					sNetId		:= AMSNetId,
					sPathName	:= CONCAT(Path,FileName),
					nMode		:= Mode ,
					ePath		:= (* Default *),
					bExecute	:= TRUE,
					tTimeout	:= Timeout,
					bBusy		=> ,
					bError		=> ,
					nErrId		=> ,
					hFile		=> );

				State 										:= 10;
			ELSE                    						
				State 										:= 10;
			END_IF                  						
		ELSE                        						
			Done											:= FALSE;
			Error											:= FALSE;
			ErrorId 										:= 0;
		END_IF

	10:
		File_Open();
		IF NOT File_Open.bBusy
		THEN
			IF File_Open.bError
			THEN
				State 										:= 99;
			ELSE
				IF File_Open.bExecute THEN hFile := File_Open.hFile; END_IF
				File_Read(
					sNetId		:= AmsNetId,
					hFile		:= hFile,
					pReadBuff	:= pBuffer,
					cbReadLen	:= Length,
					bExecute	:= TRUE,
					tTimeout	:= Timeout,
					bBusy		=> ,
					bError		=> ,
					nErrId		=> ,
					cbRead		=> ,
					bEOF		=> );

				State 										:= 20;
			END_IF
		END_IF

	20:
		File_Read(
			pReadBuff	:= pBuffer,
			cbReadLen	:= Length,
			bExecute	:= TRUE,
			cbRead		=> WorkedLen,
			bEOF		=> EOF);

		IF NOT File_Read.bBusy
		THEN
			IF File_Open.bExecute
			THEN
				File_Close(
					sNetId	:= AMSNetId,
					hFile	:= hFile,
					bExecute:= TRUE,
					tTimeout:= Timeout,
					bBusy	=> ,
					bError	=> ,
					nErrId	=> );
				State										:= 30;
			ELSE                        						
				State										:= 99;
			END_IF                      						
                                        						
		END_IF                          						
                                        						
	30:                                 						
		File_Close();                   						
		IF NOT File_Close.bBusy         						
		THEN                            						
			hFile											:= 0;
			State											:= 99;
		END_IF                          						
                                        						
	99:                                 						
		IF NOT Execute                  						
		THEN                            				
			Memfnc											:= -1;
			state 											:= 0;
		END_IF                          	
	END_CASE                            	
                                        	
	Done													:= state = 99
																AND NOT File_Read.bError
																AND NOT File_Close.bError
																AND NOT File_Open.bError;
	                                    						
	Error													:= state = 99
																AND(
																File_Read.bError
																OR File_Close.bError
																OR File_Open.bError);
	                                    						
	Busy													:= state <> 0
																AND NOT Done
																AND NOT Error;

	IF Error
	THEN
		IF File_Close.bError	THEN 	ErrorId :=  File_Close.nErrId;	END_IF
		IF File_Read.bError 	THEN	ErrorId :=  File_Read.nErrId; 	END_IF
		IF File_Open.bError		THEN	ErrorId :=  File_Open.nErrId; 	END_IF
	ELSE
		ErrorId 											:= 0;
	END_IF                              						
                                        						
	IF NOT Execute                      						
		AND state = 99                  						
	THEN                                						
		MemFnc												:=  -1;
		state 												:= 0;
	END_IF                              	
                                        	
	IF Error                            	
	THEN                                	
		MemErrorText										:= CONCAT('File_Read ErrorID: ', UDINT_TO_STRING(ErrorID));
	END_IF                              						
	                                    						
	Read													:= Busy;
END_METHOD

METHOD PUBLIC removeDir : BOOL //Return value = TRUE if busy
//required parameter
//Path
VAR_INPUT
	Execute				:	BOOL;
END_VAR
	IF Execute
	THEN
		Error												:= FALSE;
		ErrorId												:= 0;
		File_RemoveDir.bExecute 							:= TRUE;
	ELSIF NOT File_RemoveDir.bBusy      					
	THEN                                					
		Error												:=	FALSE;
		ErrorId												:= 0;
		File_RemoveDir.bExecute 							:= FALSE;
	END_IF                              					
                                        	
	MemFnc 													:= FNC_REMOVEDIR;
	THIS^.Execute											:= Execute;

	File_RemoveDir(
		sNetId		:= AMSNetId,
		sPathName	:= Path,
		ePath		:= ,
		bExecute	:= ,
		tTimeout	:= Timeout,
		bBusy		=> Busy,
		bError		=> ,
		nErrId		=> );

	Done													:= NOT File_RemoveDir.bBusy
																AND NOT File_RemoveDir.bError
																AND File_RemoveDir.bExecute;
	IF NOT Busy                         					
	THEN                                					
		IF File_RemoveDir.bExecute      					
		THEN                            					
			Error											:=	File_RemoveDir.bError;
			ErrorId											:= File_RemoveDir.nErrId;
		END_IF                          	
		IF NOT Execute                  	
		THEN                            	
			MemFnc											:=  -1;
			File_RemoveDir(bExecute := FALSE);
		END_IF
	END_IF


	IF Error
	THEN
		MemErrorText										:= CONCAT('File_RemoveDir ErrorID: ', UDINT_TO_STRING(ErrorID));
	END_IF                              					
	                                    	
	RemoveDir												:= Busy;
END_METHOD

METHOD PUBLIC rename : BOOL //Return value = TRUE if busy
//required parameter
//Path
//OldFileName
//FileName
VAR_INPUT
	Execute			:	BOOL;
END_VAR
	IF Execute
	THEN
		Error												:=	FALSE;
		ErrorId												:= 0;
		File_Rename.bExecute 								:= TRUE;
	ELSIF NOT File_Rename.bBusy         					
	THEN                                					
		Error												:=	FALSE;
		ErrorId												:= 0;
		File_Rename.bExecute 								:= FALSE;
	END_IF                              					
                                        	
	MemFnc 													:= FNC_RENAME;
	THIS^.Execute											:= Execute;

	File_Rename(
		sNetId		:= AMSNetId,
		sOldName	:= CONCAT(Path,OldFileName),
		sNewName	:= CONCAT(Path,FileName),
		ePath		:= ,
		bExecute	:=	,
		tTimeout	:=	Timeout,
		bBusy		=> Busy,
		bError		=> ,
		nErrId		=> );

	Done													:= NOT File_Rename.bBusy
																AND NOT File_Rename.bError
																AND File_Rename.bExecute;
	IF NOT Busy                         					
	THEN                                					
		IF File_Rename.bExecute         					
		THEN                            	
			Error											:=	File_Rename.bError;
			ErrorId											:= File_Rename.nErrId;
		END_IF
		IF NOT Execute
		THEN
			MemFnc											:= -1;
			File_Rename(bExecute := FALSE);
		END_IF
	END_IF


	IF Error
	THEN
		MemErrorText										:= CONCAT('File_Rename ErrorID: ', UDINT_TO_STRING(ErrorID));
	END_IF
	
	Rename													:= Busy;
END_METHOD

METHOD PUBLIC seek : BOOL //Return value = TRUE if busy
//required parameter
//Path
//SeekPos
//SeekOrigin
VAR_INPUT
	Execute			:	BOOL;
END_VAR
	IF Execute
	THEN
		Error												:=	FALSE;
		ErrorId												:= 0;
		File_Seek.bExecute 									:= TRUE;
	ELSIF NOT File_Seek.bBusy           					
	THEN                                					
		Error												:=	FALSE;
		ErrorId												:= 0;
		File_Seek.bExecute 									:= FALSE;
	END_IF                              							
	                                    	
	MemFnc 													:= FNC_SEEK;
	THIS^.Execute											:= Execute;
                                        	
	File_Seek(
		sNetId		:= AMSNetId,
		hFile		:= hFile ,
		nSeekPos	:= SeekPos,
		eOrigin		:= SeekOrigin,
		bExecute	:= ,
		tTimeout	:= Timeout,
		bBusy		=> Busy,
		bError		=> ,
		nErrId		=> );

	Done													:= NOT File_Seek.bBusy
																AND NOT File_Seek.bError
																AND File_Seek.bExecute;
	IF NOT Busy                         					
	THEN                    
		ActSeekPos											:= File_Seek.nSeekPos;           					
		IF File_Seek.bExecute           					
		THEN                            	
			Error											:=	File_Seek.bError;
			ErrorId											:= File_Seek.nErrId;
		END_IF
		IF NOT Execute
		THEN
			MemFnc											:= 1;
			File_Seek(bExecute := FALSE);
		END_IF
	END_IF


	IF Error
	THEN
		MemErrorText										:= CONCAT('File_Seek ErrorID: ', UDINT_TO_STRING(ErrorID));
	END_IF
	
	Seek													:= Busy;
END_METHOD

METHOD PUBLIC tell : BOOL //Return value = TRUE if busy
VAR_INPUT
	Execute													:	BOOL;
END_VAR
	IF Execute
	THEN
		Error												:=	FALSE;
		ErrorId												:= 0;
		File_Tell.bExecute 									:= TRUE;
	ELSIF NOT File_Tell.bBusy           					
	THEN                                					
		Error												:=	FALSE;
		ErrorId												:= 0;
		File_Tell.bExecute 									:= FALSE;
	END_IF                              					
                                        					
	MemFnc 													:= FNC_TELL;
	THIS^.Execute											:= Execute;
                                        			
	File_Tell(                          			
		sNetId		:= AMSNetId,        			
		hFile		:= hFile ,          			
		bExecute	:= ,                			
		tTimeout	:= Timeout,         			
		nSeekPos	=> ActSeekPos,      			
		bBusy		=> Busy,            			
		bError		=> ,                			
		nErrId		=> );               			
                                        			
	Done														:= NOT File_Tell.bBusy
																AND NOT File_Tell.bError
																AND File_Tell.bExecute;
	IF NOT Busy                         						
	THEN                                						
		IF File_Tell.bExecute           						
		THEN                            						
			Error												:=	File_Tell.bError;
			ErrorId												:= File_Tell.nErrId;
		END_IF                          						
		IF NOT Execute                  						
		THEN                            						
			MemFnc												:= -1;
			File_Tell(bExecute := FALSE);               	
		END_IF                                          	
	END_IF                                              	
                                                        	
                                                        	
	IF Error                                            	
	THEN                                                	
		MemErrorText											:= CONCAT('File_Tell ErrorID: ', UDINT_TO_STRING(ErrorID));
	END_IF                                              	
	                                                    	
	Tell 														:= Busy;
END_METHOD

METHOD PUBLIC write : BOOL //Return value = TRUE if busy
//required parameter
//Path
//Filename
//Mode
//pBuffer
//Length
VAR_INPUT
	Execute													:	BOOL;
END_VAR
IF pBuffer = 0 THEN
	Busy													:= NOT Error;
	Error													:= TRUE;
	ErrorId													:= E_AdsErr.DEVICE_INVALIDPARM;
	Done													:= FALSE;
	MemFnc													:= -1 ;
	RETURN;                             					
END_IF                                  					
                                        					
	MemFnc 													:= FNC_WRITE;
	THIS^.Execute											:= Execute;
                                        					
	CASE State OF                       	
	0:                                  	
		IF Execute                      	
		THEN                            	
			Done											:= FALSE;
			Error											:= FALSE;
			ErrorId 										:= 0;
			
			File_Open(bExecute := FALSE);
			File_Write(bExecute := FALSE);
			File_Close(bExecute := FALSE);	
			
			WorkedLen										:= 0;
			
			IF hFile = 0
			THEN
				File_Open(
					sNetId		:= AMSNetId,
					sPathName	:= CONCAT(Path,FileName),
					nMode		:= Mode ,
					ePath		:= (* Default *),
					bExecute	:= TRUE,
					tTimeout	:= Timeout,
					bBusy		=> ,
					bError		=> ,
					nErrId		=> ,
					hFile		=> );

				State 										:= 10;
			ELSE	                    					
				State 										:= 10;
			END_IF                      					
		ELSE                            					
			Done											:= FALSE;
			Error											:= FALSE;
			ErrorId 										:= 0;
		END_IF

	10:
		File_Open(hFile		=> hFile);

		IF NOT File_Open.bBusy
		THEN
			IF File_Open.bError
			THEN
				State 										:= 99;
			ELSE
				IF File_Open.bExecute THEN hFile := File_Open.hFile; END_IF
				File_Write(
					sNetId		:= AMSNetId,
					hFile		:= hFile,
					pWriteBuff	:= pBuffer,
					cbWriteLen	:= Length,
					bExecute	:= TRUE,
					tTimeout	:= Timeout,
					bBusy		=> ,
					bError		=> ,
					nErrId		=> ,
					cbWrite		=> );
				State 										:= 20;
			END_IF
		END_IF

	20:
		File_Write(
			pWriteBuff	:= pBuffer,
			cbWriteLen	:= Length,
			bExecute	:= TRUE,
			cbWrite		=> WorkedLen);

		IF NOT File_Write.bBusy
		THEN
			IF File_Open.bExecute
			THEN
				File_Close(
					sNetId		:= AMSNetId,
					hFile		:= hFile,
					bExecute	:= TRUE,
					tTimeout	:= Timeout,
					bBusy		=> ,
					bError		=> ,
					nErrId		=> );
				State										:= 30;
			ELSE  //Exit without closing the file as the file was opended externaly                     					
				State										:= 99;
			END_IF                  					
		ELSE                            					
			;                           					
		END_IF                          					
                                        	
	30:                                 	
		File_Close();                   	
		IF NOT File_Close.bBusy         	
		THEN                       	
			hFile											:= 0;
			State											:= 99;
		END_IF

	99:
		IF NOT Execute
		THEN	
			Memfnc											:= -1;
			state 											:= 0;
		END_IF
	END_CASE

	Done													:= state = 99
																AND NOT File_Write.bError
																AND NOT File_Close.bError
																AND NOT File_Open.bError;
                                    						
	Error													:= state = 99
																AND(
																File_Write.bError
																OR File_Close.bError
																OR File_Open.bError);
                                    						
	Busy													:= state <> 0
																AND NOT Done
																AND NOT Error;
                                    					
	IF Error
	THEN
		IF File_Close.bError 	THEN 	ErrorId :=  File_Close.nErrId;	END_IF
		IF File_Write.bError 	THEN 	ErrorId :=  File_Write.nErrId;	END_IF
		IF File_Open.bError 	THEN 	ErrorId :=  File_Open.nErrId; 	END_IF
	ELSE
		ErrorId 											:= 0;
	END_IF                          						
                                    						
	IF NOT Execute                  						
		AND state = 99              						
	THEN                            						
		MemFnc												:=  -1;
		state 												:= 0;
	END_IF                          						
                                    	
	IF Error                        	
	THEN                            	
		MemErrorText										:= CONCAT('File_Write ErrorID: ', UDINT_TO_STRING(ErrorID));
	END_IF                          	
	                                	
	Write													:= Busy;
END_METHOD

END_FUNCTION_BLOCK

// POUs/FileHandling/Basic/ReadDirSimple
{attribute 'no_check'}
//List down all files founded in a directory - specified by file type if needed 
FUNCTION_BLOCK ReadDirSimple EXTENDS FbBase
VAR_OUTPUT CONSTANT
	MIN_ENTRYS												:	INT := 1;	
	MAX_ENTRYS												:	INT := PARAM.READ_DIR_SIMPLE_MAX_ENTRYS;	//see library parameter to customize parameter	
	MAX_STRING_LEN											:	INT := PARAM.READ_DIR_SIMPLE_MAX_STRING_LEN;//see library parameter to customize parameter
END_VAR            										  										
VAR_INPUT           										
	AMSNetId												:	T_AmsNetId; //AMS Net Id
	Timeout													:	TIME := DEFAULT_ADS_TIMEOUT; //ADS Timeout Default 3s 
	Path													:	T_MaxString; // \\PC-Name\Folder\ C:\Folder\
	File													:	STRING(MAX_STRING_LEN) := '*.*'; // *.xml / *.txt
END_VAR
VAR_OUTPUT
	NoOfFiles												:	INT; //Number of files found in folder 
	EoE														:	BOOL; //end of enumeration - No more files in folder
	Entry													:	ARRAY[MIN_ENTRYS..MAX_ENTRYS] OF STRING(MAX_STRING_LEN); //List of file names
END_VAR
VAR
(* internal used variables ************************************************************)

(* trigger ****************************************************************************)	

(* function-block instances ***********************************************************)
	EnumFindFileEntry										:	FB_EnumFindFileEntry;
END_VAR


(* Sequence ****************************************)
	rtExecute(CLK := Execute);
	CASE state OF 
	0:	
		Busy												:= FALSE;
		IF NOT Execute
		THEN
			Done											:= FALSE;
			Error											:= FALSE;
			ErrorId											:= 0;
		ELSIF rtExecute.Q
		THEN
			EnumFindFileEntry(bExecute := FALSE, sNetId := AMSNetId, tTimeout := Timeout, sPathName := CONCAT(Path,File));
			Busy											:= TRUE;
			Done											:= FALSE;
			Error											:= FALSE;
			ErrorId											:= 0;
			NoOfFiles										:= 0;
			MEMSET(ADR(Entry),0,SIZEOF(Entry));
			state											:= State + 1;
		END_IF 
	
	1: //read first entry
		EnumFindFileEntry(bExecute := TRUE ,eCmd := eEnumCmd_First );
		state												:= State + 1;

	2: //read entrys
		EnumFindFileEntry(bExecute := TRUE);
		IF NOT EnumFindFileEntry.bBusy
		THEN
			IF NOT EnumFindFileEntry.bError
			THEN
				IF EnumFindFileEntry.bEOE		
				THEN
					Busy									:= FALSE;
					Done									:= TRUE;	
					state									:= 0;
					
				ELSIF NOT EnumFindFileEntry.stFindFile.fileAttributes.bDirectory
				THEN
					NoOfFiles								:= LIMIT(MIN_ENTRYS, NoOfFiles + 1 ,MAX_ENTRYS);
					Entry[NoOfFiles]						:= EnumFindFileEntry.stFindFile.sFileName;
					
					IF EnumFindFileEntry.bEOE
					THEN
						EoE									:= TRUE;
						Busy								:= FALSE;
						Done								:= TRUE;
						state								:= 0;
					ELSIF NoOfFiles >= MAX_ENTRYS
					THEN
						state								:= 3;
					ELSE
						; //Continue with next cycle					
					END_IF		
					
				END_IF
				EnumFindFileEntry(bExecute := FALSE ,eCmd := eEnumCmd_Next);
			ELSE
				Busy										:= FALSE;
				Done										:= FALSE;
				Error										:= TRUE;
				ErrorId										:= EnumFindFileEntry.nErrID;
				state										:= 0;
			END_IF		
		END_IF
		
	3: //End search
		EnumFindFileEntry(bExecute := TRUE ,eCmd := eEnumCmd_Abort);
		IF NOT EnumFindFileEntry.bBusy
		THEN
			Busy											:= FALSE;
			Done											:= NOT EnumFindFileEntry.bError;
			Error											:= NOT Done;
			ErrorId											:= EnumFindFileEntry.nErrID;
			state											:= 0;		
		END_IF
	
	END_CASE

(*************************************************************************)

END_FUNCTION_BLOCK

// POUs/FileHandling/Basic/ReadDirSimpleExt
{attribute 'no_check'}
//List down all files and it's information founded in a directory - specified by file type if needed 
FUNCTION_BLOCK ReadDirSimpleExt EXTENDS FbBase
VAR_OUTPUT CONSTANT
	MIN_ENTRYS												:	INT := 1;	
	MAX_ENTRYS												:	INT := PARAM.READ_DIR_SIMPLE_MAX_ENTRYS;	//see library parameter to customize parameter	
	MAX_STRING_LEN											:	INT := PARAM.READ_DIR_SIMPLE_MAX_STRING_LEN;//see library parameter to customize parameter
END_VAR            										  										
VAR_INPUT           										
	AMSNetId												:	T_AmsNetId; //AMS Net Id
	Timeout													:	TIME := DEFAULT_ADS_TIMEOUT; //ADS Timeout Default 3s 
	Path													:	T_MaxString; // \\PC-Name\Folder\ C:\Folder\
	File													:	STRING := '*.*'; // *.xml / *.txt
END_VAR
VAR_OUTPUT
	NoOfFiles												:	INT; //Number of files found in folder and sub folder
	EoE														:	BOOL; //end of enumeration - No more files in folder
	Entrys													:	ARRAY[MIN_ENTRYS..MAX_ENTRYS] OF ST_FindFileEntry; //List of file structures
END_VAR
VAR
(* internal used variables ************************************************************)
	
(* trigger ****************************************************************************)	

(* function-block instances ***********************************************************)
	EnumFindFileEntry										:	FB_EnumFindFileEntry;
END_VAR


(* Sequence ****************************************)
	rtExecute(CLK := Execute);
	CASE state OF 
	0:	
		Busy												:= FALSE;
		IF NOT Execute
		THEN
			Done											:= FALSE;
			Error											:= FALSE;
			ErrorId											:= 0;
		ELSIF rtExecute.Q
		THEN
			EnumFindFileEntry(bExecute := FALSE, sNetId := AMSNetId, tTimeout := Timeout, sPathName := CONCAT(Path,File));
			Busy											:= TRUE;
			Done											:= FALSE;
			Error											:= FALSE;
			ErrorId											:= 0;
			NoOfFiles										:= 0;
			MEMSET(ADR(Entrys),0,SIZEOF(Entrys));
			state											:= State + 1;
		END_IF 
	
	1: //read first entry
		EnumFindFileEntry(bExecute := TRUE ,eCmd := eEnumCmd_First );
		state												:= State + 1;

	2: //read entrys
		EnumFindFileEntry(bExecute := TRUE);
		IF NOT EnumFindFileEntry.bBusy
		THEN
			IF NOT EnumFindFileEntry.bError
			THEN
				IF EnumFindFileEntry.bEOE		
				THEN
					Busy									:= FALSE;
					Done									:= TRUE;	
					state									:= 0;
					
				ELSIF NOT EnumFindFileEntry.stFindFile.fileAttributes.bDirectory
				THEN
					NoOfFiles								:= LIMIT(MIN_ENTRYS, NoOfFiles + 1 ,MAX_ENTRYS);
					Entrys[NoOfFiles]						:= EnumFindFileEntry.stFindFile;
					
					IF EnumFindFileEntry.bEOE
					THEN
						EoE									:= TRUE;
						Busy								:= FALSE;
						Done								:= TRUE;
						state								:= 0;
					ELSIF NoOfFiles >= MAX_ENTRYS
					THEN
						state								:= 3;
					ELSE
						; //Continue with next cycle					
					END_IF		
					
				END_IF
				EnumFindFileEntry(bExecute := FALSE ,eCmd := eEnumCmd_Next);
			ELSE
				Busy										:= FALSE;
				Done										:= FALSE;
				Error										:= TRUE;
				ErrorId										:= EnumFindFileEntry.nErrID;
				state										:= 0;
			END_IF		
		END_IF
		
	3: //End search
		EnumFindFileEntry(bExecute := TRUE ,eCmd := eEnumCmd_Abort);
		IF NOT EnumFindFileEntry.bBusy
		THEN
			Busy											:= FALSE;
			Done											:= NOT EnumFindFileEntry.bError;
			Error											:= NOT Done;
			ErrorId											:= EnumFindFileEntry.nErrID;
			state											:= 0;		
		END_IF
	
	END_CASE

(*************************************************************************)

END_FUNCTION_BLOCK

// POUs/FileHandling/TF6421-XmlServer/XmlReadWrite
{attribute 'no_check'}
//Wrapper for functions of TF6421 XML-Server
//based on TF6421 - required lib: Tc2_XmlDataSvr - see Beckhoff documentation for more information
FUNCTION_BLOCK XmlReadWrite EXTENDS FbBase
VAR_OUTPUT CONSTANT
	FNC_READ												:	INT := 0; //Read data from XML
	FNC_WRITE												:	INT := 1; //Create XML if not exist and wite data into file
END_VAR             										
VAR_INPUT           										
	Fnc														:	INT (FNC_READ..FNC_WRITE) := FNC_READ; //See output constants for possible parameter
	NetId													: 	T_AmsNetId := ''; //Ams Net ID
	Mode													: 	WORD := XMLSRV_ADDMISSING; // XMLSRV_SKIPMISSING or XMLSRV_ADDMISSING;
	pSymAddr												: 	PVOID := 0;	//Pointer to target variable to read or write data 
	SymSize													:	UDINT := 0;	//Size of variable/structure
	FilePath												:	T_MaxString := 'C:\'; // \\PCName\Folder\test.xml
	FileName												:	T_MaxString := 'data.xml'; // \\PCName\Folder\test.xml
	XPath													:	T_MaxString := '/dataentry/data'; // XML tag name/adress to access all or specified data insite the file. Array access->CONCAT('/Datentry/Step[@index="',CONCAT(DINT_TO_STRING(AktStep),'"]')); 										
	Timeout													: 	TIME := T#60S;
END_VAR             										
VAR_OUTPUT          										
END_VAR             	
VAR                 	
(* Local variables ************************************************************)
	MemFnc													:	INT := -1;
	
(* Trigger *****************************************************************)

(* Timer ******************************************************************)

(* Fcuntion blocks ***************************************************************)
	XmlSrvRead 												: 	FB_XmlSrvRead;
	XmlSrvWrite 											: 	FB_XmlSrvWrite;

(* Dummys **********************************************************)

END_VAR

	(* XML Read/Write														V2.0		*)
	(************************************************************************************)

(* Execute ***************************************************************************************)
	rtExecute(CLK := Execute);
	IF rtExecute.Q
		AND MemFnc < 0
	THEN
		MemFnc 												:= SEL(Fnc = FNC_WRITE, FNC_READ , FNC_WRITE) ;
		Busy												:= TRUE;
		Done												:= FALSE;
		Error												:= FALSE;
		ErrorID												:= 0;
	END_IF

(* Call Method ***********************************************************************************)
	CASE MemFnc OF
	FNC_READ:
		Read(
			Execute	:= Execute);
	
	FNC_WRITE:
		Write(			
			Execute	:= Execute);
			
	-1:
		IF NOT Execute
		THEN
			Busy											:= FALSE;
			Done											:= FALSE;
			Error											:= FALSE;
			ErrorID											:= 0;
		END_IF                              				
	ELSE                                    				
		Busy												:= FALSE;
		Done												:= FALSE;
		Error												:= Execute;
		ErrorID												:= E_AdsErr.DEVICE_INVALIDPARM;
	END_CASE

(*************************************************************************************************)

METHOD PUBLIC read : BOOL //Return value = TRUE if busy
//required parameter
//pSymAddr
//SymSize
//FilePath
//XPath
VAR_INPUT
	Execute													:	BOOL;
END_VAR
IF pSymAddr = 0 THEN
	Busy													:= NOT Error;
	Error													:= TRUE;
	ErrorId													:= E_AdsErr.DEVICE_INVALIDPARM;
	Done													:= FALSE;
	MemFnc													:= -1 ;
	RETURN;
END_IF

	IF Execute
	THEN
		Error												:=	FALSE;
		ErrorId												:= 0;
		XmlSrvRead.bExecute 								:= TRUE;
	ELSIF NOT XmlSrvRead.bBusy      						
	THEN                            						
		Error												:=	FALSE;
		ErrorId												:= 0;
		XmlSrvRead.bExecute 								:= FALSE;
                                    						
	END_IF                          						
                                    	
	MemFnc													:= FNC_READ;
	                                						
	THIS^.Execute											:= Execute;
                                    						
	XmlSrvRead(                    	
		sNetId		:= NetId,
		ePath		:= ,(* Default *)
		nMode		:= XMLSRV_SKIPMISSING, 
		pSymAddr	:= pSymAddr,
		cbSymSize	:= SymSize,
		sFilePath	:= CONCAT(FilePath,FileName),
		sXPath		:= XPath,
		bExecute	:=  ,
		tTimeout	:= Timeout,
		bBusy		=> Busy,
		bError		=> ,
		nErrId		=> );

	Done													:= NOT XmlSrvRead.bBusy
																AND NOT XmlSrvRead.bError
																AND XmlSrvRead.bExecute;
                                        				
	IF NOT Busy
	THEN
		IF XmlSrvRead.bExecute
		THEN
			Error											:=	XmlSrvRead.bError;
			ErrorId											:= XmlSrvRead.nErrId;
		END_IF
		IF NOT Execute
		THEN
			MemFnc											:= -1 ;
			XmlSrvRead(bExecute := FALSE);
		END_IF
	END_IF
	
	Read													:= Busy;
END_METHOD

METHOD PUBLIC write : BOOL //Return value = TRUE if busy
//required parameter
//pSymAddr
//SymSize
//FilePath
//XPath
VAR_INPUT
	Execute				:	BOOL;
END_VAR
IF pSymAddr = 0 
THEN
	Busy													:= NOT Error;
	Error													:= TRUE;
	ErrorId													:= E_AdsErr.DEVICE_INVALIDPARM;
	Done													:= FALSE;
	MemFnc													:= -1 ;
	RETURN;
END_IF

	IF Execute
	THEN
		Error												:=	FALSE;
		ErrorId												:= 0;
		XmlSrvWrite.bExecute 								:= TRUE;
	ELSIF NOT XmlSrvWrite.bBusy     						
	THEN                            						
		XmlSrvWrite.bExecute								:= FALSE;
		Error												:=	FALSE;
		ErrorId												:= 0;
	END_IF                          						
                                    						
	MemFnc													:= FNC_WRITE;
	                                						
	THIS^.Execute											:= Execute;
                                    	
	XmlSrvWrite(
		sNetId		:= NetId,
		ePath		:= ,(* Default *)
		nMode		:= Mode,
		pSymAddr	:= pSymAddr,
		cbSymSize	:= SymSize,
		sFilePath	:= CONCAT(FilePath,FileName),
		sXPath		:= XPath,
		bExecute	:= ,
		tTimeout	:= Timeout,
		bBusy		=> Busy,
		bError		=> ,
		nErrId		=> );

	Done													:= NOT XmlSrvWrite.bBusy
																AND NOT XmlSrvWrite.bError
																AND XmlSrvWrite.bExecute;
                                        					
	IF NOT Busy
	THEN
		IF XmlSrvWrite.bExecute
		THEN
			Error											:=	XmlSrvWrite.bError;
			ErrorId											:= XmlSrvWrite.nErrId;
		END_IF
		IF NOT Execute
		THEN
			MemFnc											:= -1;
			XmlSrvWrite(bExecute := FALSE);
		END_IF
	END_IF

	Write													:= Busy;
END_METHOD

END_FUNCTION_BLOCK

